# B&R Automation Studio project A2019059_Linka_Power_CP (part 13)

#### RFID.fun - Exported functions and function blocks
```iecst
FUNCTION_BLOCK TP_Init (*TODO: Add your comment here*)
	VAR_INPUT
		Enable : BOOL; (*Add your parameter comment*)
	END_VAR
	VAR_OUTPUT
		Ident : ARRAY[0..10] OF UDINT;
		Error : BOOL;
		ErrorID : UDINT;
		Busy : BOOL;
		Done : BOOL;
	END_VAR
	VAR
		StepInit : USINT;
		USBNodeListGetFuB : UsbNodeListGet;
		status : status;
		usbNodeList : ARRAY[0..31] OF UDINT;
		i : UINT;
		USBNodeGetFuB : UsbNodeGet;
		usbDevice : ARRAY[0..10] OF usbNode_typ;
		StringDevice : ARRAY[0..10] OF STRING[30];
	END_VAR
END_FUNCTION_BLOCK
(********************************************************************
 * COPYRIGHT -- Bernecker + Rainer
 ********************************************************************
 * Library: RFID
 * File: RFID.fun
 * Author: houx
 * Created: March 25, 2009
 ********************************************************************
 * Functions and function blocks of library RFID
 ********************************************************************)

FUNCTION_BLOCK TP_Info (*TODO: Add your comment here*)
	VAR_INPUT
		Enable : BOOL; (*Add your parameter comment*)
		Ident : UDINT;
	END_VAR
	VAR_OUTPUT
		Busy : BOOL;
		Done : BOOL;
		Error : BOOL;
		ErrorID : UDINT;
		Info : Info;
	END_VAR
	VAR
		Stepstatus : USINT;
		WriteData : ARRAY[0..255] OF USINT;
		FrameWriteStruct : FRM_write;
		status : status;
		FrameReadStruct : FRM_read;
		ReadBuffer : UDINT;
		ReadBufferLength : UINT;
		ReadData : ARRAY[0..255] OF USINT;
		FrameReleaseBufferStruct : FRM_rbuf;
		ID : ARRAY[0..9] OF USINT;
		StackLevel : ARRAY[0..1] OF USINT;
		KeyType : ARRAY[0..3] OF USINT;
		AN : ARRAY[0..2] OF USINT;
		sendbuffer : UDINT;
		FrameGetBufferStruct : FRM_gbuf;
		sendbufferlength : UINT;
		FrameReleaseOutputBufferStruct : FRM_robuf;
		FrameXOpenStruct : FRM_xopen;
	END_VAR
END_FUNCTION_BLOCK

FUNCTION_BLOCK TP_Unlock (*TODO: Add your comment here*)
	VAR_INPUT
		Enable : BOOL; (*Add your parameter comment*)
		Ident : UDINT;
		Data : UDINT;
	END_VAR
	VAR_OUTPUT
		Busy : BOOL;
		Error : BOOL;
		ErrorID : UDINT;
		Done : BOOL;
	END_VAR
	VAR
		StepType : USINT;
		WriteData : ARRAY[0..255] OF USINT;
		FrameWriteStruct : FRM_write;
		status : status;
		FrameReadStruct : FRM_read;
		ReadBuffer : UDINT;
		ReadBufferLength : UINT;
		ReadData : ARRAY[0..255] OF USINT;
		FrameReleaseBufferStruct : FRM_rbuf;
		string1 : STRING[20];
		string2 : STRING[10];
		CMD : UDINT;
		StepWrite : USINT;
		ERROR : ARRAY[0..2] OF USINT;
		AN : ARRAY[0..2] OF USINT;
		FrameGetBufferStruct : FRM_gbuf;
		sendbuffer : UDINT;
		sendbufferlength : UINT;
		FrameReleaseOutputBufferStruct : FRM_robuf;
		FrameXOpenStruct : FRM_xopen;
		TypeOK : BOOL;
	END_VAR
END_FUNCTION_BLOCK

FUNCTION_BLOCK TP_Lock (*TODO: Add your comment here*)
	VAR_INPUT
		Enable : BOOL; (*Add your parameter comment*)
		Ident : UDINT;
	END_VAR
	VAR_OUTPUT
		Busy : BOOL;
		ErrorID : UDINT;
		Error : BOOL;
		Done : BOOL;
	END_VAR
	VAR
		WriteData : ARRAY[0..255] OF USINT;
		FrameWriteStruct : FRM_write;
		status : status;
		FrameReadStruct : FRM_read;
		ReadBuffer : UDINT;
		ReadData : ARRAY[0..255] OF USINT;
		ReadBufferLength : UINT;
		FrameReleaseBufferStruct : FRM_rbuf;
		StepLOCK : USINT;
		AN : ARRAY[0..2] OF USINT;
		ERROR : ARRAY[0..2] OF USINT;
		TypeOK : BOOL;
		StepType : USINT;
		FrameGetBufferStruct : FRM_gbuf;
		sendbufferlength : UINT;
		sendbuffer : UDINT;
		FrameReleaseOutputBufferStruct : FRM_robuf;
		FrameXOpenStruct : FRM_xopen;
	END_VAR
END_FUNCTION_BLOCK

FUNCTION_BLOCK TP_PWProtect (*TODO: Add your comment here*)
	VAR_INPUT
		Enable : BOOL; (*Add your parameter comment*)
		Ident : UDINT;
		Data : UDINT;
	END_VAR
	VAR_OUTPUT
		Busy : BOOL;
		Error : BOOL;
		ErrorID : UDINT;
		Done : BOOL;
	END_VAR
	VAR
		TypeOK : BOOL;
		StepType : USINT;
		WriteData : ARRAY[0..255] OF USINT;
		FrameWriteStruct : FRM_write;
		status : status;
		FrameReadStruct : FRM_read;
		ReadBuffer : UDINT;
		ReadBufferLength : UINT;
		ReadData : ARRAY[0..255] OF USINT;
		FrameReleaseBufferStruct : FRM_rbuf;
		string1 : STRING[20];
		string2 : STRING[20];
		CMD : UDINT;
		StepWrite : USINT;
		AN : ARRAY[0..2] OF USINT;
		ERROR : ARRAY[0..2] OF USINT;
		FrameGetBufferStruct : FRM_gbuf;
		sendbuffer : UDINT;
		sendbufferlength : UINT;
		FrameReleaseOutputBufferStruct : FRM_robuf;
		FrameXOpenStruct : FRM_xopen;
	END_VAR
END_FUNCTION_BLOCK

FUNCTION_BLOCK TP_OnOff (*TODO: Add your comment here*)
	VAR_INPUT
		Enable : BOOL; (*Add your parameter comment*)
		Ident : UDINT;
		Mode : BOOL;
	END_VAR
	VAR_OUTPUT
		Error : BOOL;
		ErrorID : UDINT;
		Busy : BOOL;
		Done : BOOL;
	END_VAR
	VAR
		StepOnOff : USINT;
		WriteData : ARRAY[0..255] OF USINT;
		FrameWriteStruct : FRM_write;
		status : status;
		FrameReadStruct : FRM_read;
		ReadBuffer : UDINT;
		ReadBufferLength : UINT;
		ReadData : ARRAY[0..255] OF USINT;
		FrameReleaseOutputBufferStruct : FRM_robuf;
		AN : ARRAY[0..2] OF USINT;
		FrameGetBufferStruct : FRM_gbuf;
		sendbuffer : UDINT;
		sendbufferlength : UINT;
		FrameReleaseBufferStruct : FRM_rbuf;
		FrameXOpenStruct : FRM_xopen;
		FRM_close_0 : FRM_close;
	END_VAR
END_FUNCTION_BLOCK

FUNCTION_BLOCK TP_Crc (*TODO: Add your comment here*)
	VAR_INPUT
		Enable : BOOL; (*Add your parameter comment*)
		Ident : UDINT;
		Mode : BOOL;
	END_VAR
	VAR_OUTPUT
		Error : BOOL;
		ErrorID : UDINT;
		Busy : BOOL;
		Done : BOOL;
	END_VAR
	VAR
		WriteData : ARRAY[0..255] OF USINT;
		FrameWriteStruct : FRM_write;
		FrameReadStruct : FRM_read;
		ReadBuffer : UDINT;
		ReadData : ARRAY[0..255] OF USINT;
		ReadBufferLength : UINT;
		FrameReleaseBufferStruct : FRM_rbuf;
		status : status;
		StepCRC : USINT;
		AN : ARRAY[0..2] OF USINT;
		FrameGetBufferStruct : FRM_gbuf;
		sendbuffer : UDINT;
		sendbufferlength : UINT;
		FrameReleaseOutputBufferStruct : FRM_robuf;
		FrameXOpenStruct : FRM_xopen;
		FRM_close_0 : FRM_close;
	END_VAR
END_FUNCTION_BLOCK

FUNCTION_BLOCK TP_Write (*TODO: Add your comment here*)
	VAR_INPUT
		Enable : BOOL; (*Add your parameter comment*)
		RegNr : USINT;
		Data : UDINT;
		Ident : UDINT;
	END_VAR
	VAR_OUTPUT
		Busy : BOOL;
		Error : BOOL;
		ErrorID : UDINT;
		Done : BOOL;
	END_VAR
	VAR
		CMD : UDINT;
		WriteData : ARRAY[0..255] OF USINT;
		StepWrite : USINT;
		FrameWriteStruct : FRM_write;
		status : status;
		CommandReady : BOOL;
		ReadBuffer : UDINT;
		FrameReleaseBufferStruct : FRM_rbuf;
		ReadBufferLength : UINT;
		FrameReadStruct : FRM_read;
		ReadData : ARRAY[0..255] OF USINT;
		string1 : STRING[30];
		string2 : STRING[30];
		StepType : USINT;
		TypeOK : BOOL;
		string3 : STRING[10];
		AN : ARRAY[0..2] OF USINT;
		ERROR : ARRAY[0..2] OF USINT;
		KeyType : ARRAY[0..3] OF USINT;
		FrameGetBufferStruct : FRM_gbuf;
		sendbuffer : UDINT;
		sendbufferlength : UINT;
		FrameReleaseOutputBufferStruct : FRM_robuf;
		FrameXOpenStruct : FRM_xopen;
	END_VAR
END_FUNCTION_BLOCK

FUNCTION_BLOCK TP_Read (*TODO: Add your comment here*)
	VAR_INPUT
		Enable : BOOL; (*Add your parameter comment*)
		RegNr : USINT;
		Ident : UDINT;
	END_VAR
	VAR_OUTPUT
		Done : BOOL;
		Error : BOOL;
		ErrorID : UDINT;
		Busy : BOOL;
		Data : UDINT;
	END_VAR
	VAR
		CommandReady : BOOL;
		WriteData : ARRAY[0..255] OF USINT;
		status : status;
		ReadBuffer : UDINT;
		ReadBufferLength : UINT;
		ReadData : ARRAY[0..255] OF USINT;
		FrameReadStruct : FRM_read;
		data : ARRAY[0..19] OF USINT;
		FrameReleaseBufferStruct : FRM_rbuf;
		FrameWriteStruct : FRM_write;
		TypeOK : BOOL;
		StepType : USINT;
		KeyType : ARRAY[0..3] OF USINT;
		AN : ARRAY[0..2] OF USINT;
		ERROR : ARRAY[0..2] OF USINT;
		FrameGetBufferStruct : FRM_gbuf;
		sendbuffer : UDINT;
		sendbufferlength : UINT;
		FrameReleaseOutputBufferStruct : FRM_robuf;
		FrameXOpenStruct : FRM_xopen;
		StepREAD : USINT;
	END_VAR
END_FUNCTION_BLOCK
```

#### TP_Init.st
```iecst
(********************************************************************
 * COPYRIGHT -- Bernecker + Rainer
 ********************************************************************
 * Library: RFID
 * File: TP_Init.st
 * Author: houx
 * Created: March 25, 2009
 *****************************************************************
FuB: 			TP_Init
*****************************************************************
Discription:
	USB Interface:	This FuB find the Transponder Reader(USB) in the Target and read out the Interface Ident.
								Interface Ident ist required for all other FuBs in RFID Library.
								This FuB can work without any transponder in the range of Reader.
	serial Interface:	This FuB is not used to find a serial interface transponder reader
Parameter:
	Input:
		Enable(BOOL)	: The function block is only executed when enable is <> 0
	Output:
		Error(BOOL)		: Error = 0 (No Error) Error = 1(see ErrorID)
		ErrorID(UDINT)	: Number and Description in Error Table
		Busy(BOOL)		: Fub working on
		Ident(UDINT)	: Interface ID
		Done(BOOL)		: success, if TRUE
Author:	Xiaoguang Hou
		B&R Eggelsberg

History: 	V1.00.0 - 02 Sep 2008 first create
				V3.00.0 - 25 Mar 2009  update for serial interface transponder reader and created under AS3.0

*****************************************************************

 ********************************************************************
 * Implementation of library RFID
 ********************************************************************)

FUNCTION_BLOCK TP_Init

(*------------------------------------------------------	Start	---------------------------------------------------------*)
IF Enable = TRUE THEN
	IF (Done = FALSE) AND (Error = FALSE) THEN
		Busy	:=	TRUE;
		CASE StepInit OF
	(*	------------------------------------------------	search usb device	---------------------------------------------*)
			SEARCHTPLIST :
				USBNodeListGetFuB(enable := TRUE,pBuffer := ADR(usbNodeList),bufferSize := SIZEOF(usbNodeList));
				status.GetUsbList				:=USBNodeListGetFuB.status;
				IF status.GetUsbList = 0  THEN
					StepInit					:=SEARCHTP;
					USBNodeListGetFuB.enable 	:= FALSE;
				END_IF
	(*	------------------------------------------------	if Error ?show ErrorID	----------------------------------------------------*)
				IF (status.GetUsbList <> 0) AND (status.GetUsbList <> 65535) THEN
					StepInit 	:= SEARCHTPLIST;
					Error		:= TRUE;
					Busy		:= FALSE;
					ErrorID		:= status.GetUsbList;
				END_IF
	(*	----------------------------------------------- usb device identizification , a Transponder ? get the deviceID----------------------*)
			SEARCHTP:
				USBNodeGetFuB(enable := TRUE,nodeId := usbNodeList[i],pBuffer := ADR(usbDevice[i]),bufferSize :=256 (*SIZEOF(usbDevice)*));
				status.GetUsbNode := USBNodeGetFuB.status;
				IF  status.GetUsbNode = 0 THEN
					IF	(usbDevice[i].vendorId = TRANSPONDER_VENDOR_ID) AND (usbDevice[i].productId = TRANSPONDER_PRODUCT_ID) AND (usbDevice[i].bcdDevice = TRANSPONDER_BCD) THEN
						strcpy(ADR(StringDevice[i]),ADR(usbDevice[i].ifName));
						Ident[i]				:= ADR(StringDevice[i]);
						Done                    := TRUE;
						Busy                    := FALSE;
						USBNodeGetFuB.enable 	:= FALSE;
						i						:= i+1;
						IF i= USBNodeListGetFuB.listNodes THEN
							i           	        := 0;
							StepInit				:= SEARCHTPLIST;
						END_IF
					ELSE
						i						:= i+1;
					END_IF
				ELSIF status.GetUsbNode = 65535 THEN
					StepInit				:=SEARCHTP;
				ELSE
					StepInit :=  SEARCHTPLIST;
					Error 	 :=  TRUE;
					Busy     :=  FALSE;
					ErrorID  :=  status.GetUsbNode;
				END_IF
		END_CASE
	END_IF
	(*	------------------------------------------------	Not Enable, set parameters FALSE	----------------------------------------------------*)
ELSE
	Busy	:=	FALSE;
	Error	:=	FALSE;
	Done	:=	FALSE;
	ErrorID	:=	FALSE;
END_IF
(*	------------------------------------------------	end	----------------------------------------------------*)
END_FUNCTION_BLOCK
```

#### TP_Info.st
```iecst
(********************************************************************
 * COPYRIGHT -- Bernecker + Rainer
 ********************************************************************
 * Library: RFID
 * File: TP_Info.st
 * Author: houx
 * Created: March 25, 2009
*****************************************************************
FuB: 			TP_Info
;*****************************************************************
Discription:
	This FuB can be used to output the Transponder Type, the stack lever and HW/SW	versions.
	This Fub can only work, if any Transponder in the range of Reader.
	Type			: 4150 R/W or 4102 R
	Stack level		: stack level in transponder memory
	HW/SW version	:	guarantees that your application software is being operated with the correct readers.
Parameter:
			Input: 		Enable(BOOL)	:	The function block is only executed when enable is <> 0
				   			Ident(UDINT)	:	Interface Ident from TP_Init.
			Output: 	Error(BOOL)		:	Error = 0 (No Error) Error = 1(see ErrorID)
							ErrorID(UDINT)	:	Number and Description in Error Table
							Busy(BOOL)		:	if TRUE , Fub working on.
							Done(BOOL)		:	if TRUE, success
							Info(Info)		:	Structure with Type, ID and Stacklevel.
Author:				Xiaoguang Hou
							B&R Eggelsberg
;History:	V1.00.0 - 02 Sep 2008 : first create
				V3.00.0 - 25 Mar 2009 : update for serial interface transponder and created under AS3.0
 ********************************************************************
 * Implementation of library RFID
 ********************************************************************)

FUNCTION_BLOCK TP_Info
(*--------------------------------------	start	----------------------------*)
IF (Enable = 1) THEN
	IF ((Done = 0) AND (Error = 0)) THEN
		Busy	:=	TRUE;
		CASE Stepstatus OF
(*	------------------------------------------------	open the interface, get the internal Ident	----------------------------------------------------*)
			OPEN:
				FrameXOpenStruct(enable := 1,device := Ident);
				status.XOPEN 			:= FrameXOpenStruct.status;
				IF (status.XOPEN = 0) THEN
					Stepstatus          := TYPEWRITE ;
					FrameXOpenStruct.enable := FALSE;
				ELSE
					Stepstatus          := OPEN ;
					Error               := TRUE;
					ErrorID             := status.XOPEN;
					Busy                := 0;
				END_IF
			TYPEWRITE:
				memset(ADR(WriteData),0,SIZEOF(WriteData));
				strcpy(ADR(WriteData),ADR('tag,0,0,#crc$R$L'));
				FrameGetBufferStruct(enable:= 1, ident:= FrameXOpenStruct.ident);
				sendbuffer					:= FrameGetBufferStruct.buffer;
				sendbufferlength		:= FrameGetBufferStruct.buflng;
				status.GetBuffer		:= FrameGetBufferStruct.status;
				IF	(status.GetBuffer = 0)	THEN
					memcpy(sendbuffer,ADR(WriteData),sendbufferlength);
					FrameWriteStruct(enable := 1, ident := FrameXOpenStruct.ident, buffer := sendbuffer,buflng := strlen(ADR(WriteData)));
					status.WRITE 			:=	FrameWriteStruct.status;
				  	IF (status.WRITE <> 0) THEN
						FrameReleaseOutputBufferStruct(enable:=1,ident:=FrameXOpenStruct.ident,buffer:=sendbuffer,buflng:=strlen(ADR(WriteData)) );
						status.RoBuffer			:= FrameReleaseOutputBufferStruct.status;
					ELSE
				    	FrameGetBufferStruct.enable	:= 0;
						FrameWriteStruct.enable := 0;
						FrameReleaseOutputBufferStruct.enable := 0;
						Stepstatus              :=	TYPEREAD;
					END_IF
				ELSE
					ErrorID 	:= status.GetBuffer;
					Error   	:= 1;
					Busy    	:= 0;
					FrameGetBufferStruct.enable	:= 0;
					Stepstatus	:= OPEN;
				END_IF
			TYPEREAD:
				FrameReadStruct(enable:=1,ident:=FrameXOpenStruct.ident);
				ReadBuffer       	:=	FrameReadStruct.buffer;
				ReadBufferLength	:=	FrameReadStruct.buflng;
				status.READ      	:=	FrameReadStruct.status;
				IF  (status.READ = 0) THEN
					memset(ADR(ReadData),0,SIZEOF(ReadData));
					memcpy(ADR(ReadData),ReadBuffer,ReadBufferLength);                   (* copy read data into read buffer *)
					FrameReadStruct.enable	:= 0;
			        FrameReleaseBufferStruct(enable:=1, ident:=FrameXOpenStruct.ident, buffer:=ReadBuffer,buflng:=ReadBufferLength);        (* release read buffer *)
			        status.ReleaseBuffer	:=FrameReleaseBufferStruct.status;
			        IF (status.ReleaseBuffer=0) THEN
				        FrameReleaseBufferStruct.enable:=0;
						AN[0]		 :=	ReadData[0];
						AN[1]		 := ReadData[1];
						AN[2]		 := ReadData[2];
						IF	(memcmp(ADR(AN),ADR('ack'),3) = 0)	THEN
							memset(ADR(KeyType),0,SIZEOF(KeyType));
							KeyType[0]   	 := ReadData[6];
							KeyType[1] 	 := ReadData[7];
							KeyType[2] 	 := ReadData[8];
							KeyType[3] 	 := ReadData[9];
							IF (memcmp(ADR(KeyType),ADR('4150'),4) = 0) THEN
								Info.Type	:=	ADR(KeyType);
								Stepstatus	:=	IDWRITE;
							ELSIF	(memcmp(ADR(KeyType),ADR('4102'),4) = 0) THEN
								Info.Type	:=	ADR(KeyType);
								Stepstatus	:=	IDWRITE;
							ELSE
								Stepstatus	:= OPEN;
								ErrorID	:=	rfidError_tag_failed; (* unknow type of transponder *)
								Error   :=	1;
								Busy    :=	0;
							END_IF
						ELSIF	(memcmp(ADR(AN),ADR('nak'),3) = 0)	THEN
							Stepstatus	:= OPEN;
							ErrorID	:=	rfidError_tag_failed; (* negativ answer *)
							Error   :=	1;
							Busy    :=	0;
						ELSE
							Stepstatus	:= OPEN;
							ErrorID	:=	rfidError_tag_failed; (* unknow answer *)
							Error   :=	1;
							Busy    :=	0;
						END_IF
					ELSE
						Stepstatus	:=	OPEN;
						Error     	:=	1;
						ErrorID   	:=	status.ReleaseBuffer;
						Busy      	:=	0;
					END_IF
				ELSE
					memset(ADR(ReadData),0,SIZEOF(ReadData));
				END_IF
			IDWRITE:
				memset(ADR(WriteData),0,SIZEOF(WriteData));
				strcpy(ADR(WriteData),ADR('id,0,#crc$R$L'));
				FrameGetBufferStruct(enable:= 1, ident:= FrameXOpenStruct.ident);
				sendbuffer				    := FrameGetBufferStruct.buffer;
				sendbufferlength		:= FrameGetBufferStruct.buflng;
				status.GetBuffer		:= FrameGetBufferStruct.status;
				IF	(status.GetBuffer = 0)	THEN
					memcpy(sendbuffer,ADR(WriteData),sendbufferlength);
					FrameWriteStruct(enable := 1, ident := FrameXOpenStruct.ident, buffer := sendbuffer,buflng := strlen(ADR(WriteData)));
					status.WRITE 			:=	FrameWriteStruct.status;

			        IF (status.WRITE <> 0) THEN
						FrameReleaseOutputBufferStruct(enable:=1,ident:=FrameXOpenStruct.ident,buffer:=sendbuffer,buflng:= strlen(ADR(WriteData)));
						status.RoBuffer			:= FrameReleaseOutputBufferStruct.status;
						IF	(status.RoBuffer <> 0)	THEN
							ErrorID	:= status.RoBuffer;
						END_IF
					ELSE
			        	FrameWriteStruct.enable := 0;
						FrameGetBufferStruct.enable	:= 0;
						FrameReleaseOutputBufferStruct.enable := 0;
						Stepstatus              :=	IDREAD;
					END_IF
				ELSE
					ErrorID 	:= status.GetBuffer;
					Error   	:= 1;
					Busy    	:= 0;
					Stepstatus	:= OPEN;
					FrameGetBufferStruct.enable	:= 0;
				END_IF

			IDREAD:
				FrameReadStruct(enable:=1,ident:=FrameXOpenStruct.ident);
				ReadBuffer       	:=	FrameReadStruct.buffer;
				ReadBufferLength	:=	FrameReadStruct.buflng;
				status.READ      	:=	FrameReadStruct.status;
				IF  (status.READ = 0) THEN
					memset(ADR(ReadData),0,SIZEOF(ReadData));
					memcpy(ADR(ReadData),ReadBuffer,ReadBufferLength);                   (* copy read data into read buffer *)
					FrameReadStruct.enable	:=	0;
			        FrameReleaseBufferStruct(enable:=1, ident:=FrameXOpenStruct.ident, buffer:=ReadBuffer,buflng:=ReadBufferLength);        (* release read buffer *)
			        status.ReleaseBuffer	:=	FrameReleaseBufferStruct.status;
			        IF (status.ReleaseBuffer=0) THEN
				        FrameReleaseBufferStruct.enable	:=	0;
				        AN[0]	:= ReadData[0];
						AN[1]	:= ReadData[1];
						AN[2]	:= ReadData[2];
				        IF	(memcmp(ADR(AN),ADR('ack'),3) = 0) THEN
				        	memset(ADR(ID),0,SIZEOF(ID));
							ID[0] 	 	:=	ReadData[6];
							ID[1] 	 	:=	ReadData[7];
							ID[2] 	 	:=	ReadData[8];
							ID[3] 	 	:=	ReadData[9];
							ID[4] 	 	:=	ReadData[11];
							ID[5] 	 	:=	ReadData[12];
							ID[6] 	 	:=	ReadData[13];
							ID[7] 	 	:=	ReadData[14];
							Info.ID   	:=	ADR(ID);
							Stepstatus  :=	STACKWRITE;
						ELSE
							Stepstatus	:= OPEN;
							Error     	:= 1;
							ErrorID   	:= rfidError_id_failed;	(* negativ answer by ask for ID *)
							Busy      	:= 0;
						END_IF
					ELSE
						Stepstatus	:= OPEN;
						Error     	:= 1;
						ErrorID   	:= status.ReleaseBuffer;
						Busy      	:= 0;
					END_IF
				ELSE
					memset(ADR(ReadData),0,SIZEOF(ReadData));
				END_IF
			STACKWRITE:
				memset(ADR(WriteData),0,SIZEOF(WriteData));
				strcpy(ADR(WriteData),ADR('stack,0,#crc$R$L'),);
				FrameGetBufferStruct(enable:= 1, ident:= FrameXOpenStruct.ident);
				sendbuffer				:= FrameGetBufferStruct.buffer;
				sendbufferlength		:= FrameGetBufferStruct.buflng;
				status.GetBuffer		:= FrameGetBufferStruct.status;
				IF	(status.GetBuffer = 0)	THEN
					memcpy(sendbuffer,ADR(WriteData),sendbufferlength);
					FrameWriteStruct(enable := 1, ident := FrameXOpenStruct.ident, buffer := sendbuffer,buflng := strlen(ADR(WriteData)));
					status.WRITE 		:=	FrameWriteStruct.status;
			        Stepstatus          :=	STACKREAD;
			        IF (status.WRITE <> 0) THEN
						FrameReleaseOutputBufferStruct(enable:=1,ident:=FrameXOpenStruct.ident,buffer:=sendbuffer,buflng:= strlen(ADR(WriteData)));
						status.RoBuffer			:= FrameReleaseOutputBufferStruct.status;
						IF	(status.RoBuffer <> 0)	THEN
							ErrorID	:= status.RoBuffer;
						END_IF
					END_IF
					FrameWriteStruct.enable :=	0;
					FrameGetBufferStruct.enable	:= 0;
					FrameReleaseOutputBufferStruct.enable := 0;
				ELSE
					ErrorID 	:= status.GetBuffer;
					Error   	:= 1;
					Busy    	:= 0;
					Stepstatus	:= OPEN;
					FrameGetBufferStruct.enable	:= 0;
				END_IF
			STACKREAD:
				FrameReadStruct(enable:=1,ident:=FrameXOpenStruct.ident);
				ReadBuffer       	:=	FrameReadStruct.buffer;
				ReadBufferLength	:=	FrameReadStruct.buflng;
				status.READ      	:=	FrameReadStruct.status;
				IF  (status.READ = 0) THEN
					memset(ADR(ReadData),0,SIZEOF(ReadData));
					memcpy(ADR(ReadData),ReadBuffer,ReadBufferLength);                   (* copy read data into read buffer *)
					FrameReadStruct.enable	:=	0;
			        FrameReleaseBufferStruct(enable:=1, ident:=FrameXOpenStruct.ident, buffer:=ReadBuffer,buflng:=ReadBufferLength);        (* release read buffer *)
			        status.ReleaseBuffer	:=	FrameReleaseBufferStruct.status;
			        IF (status.ReleaseBuffer = 0) THEN
				        FrameReleaseBufferStruct.enable	:=	0;
				        AN[0]	:= ReadData[0];
						AN[1]	:= ReadData[1];
						AN[2]	:= ReadData[2];
				        IF	(memcmp(ADR(AN),ADR('ack'),3) = 0) THEN
							memset(ADR(StackLevel),0,SIZEOF(StackLevel));
							StackLevel[0] 	  :=	ReadData[6];
							StackLevel[1] 	  :=	ReadData[7];
							Info.StackLevel :=	ADR(StackLevel);
							Stepstatus		  :=	OPEN;
							Done			  :=	1;
							Busy			  :=	0;
						ELSE
							Stepstatus	:=	OPEN;
							Error     	:=	1;
							ErrorID   	:=	rfidError_stacklevel_failed;
							Busy      	:=	0;
						END_IF
					ELSE
						Stepstatus	:=	OPEN;
						Error     	:=	1;
						ErrorID   	:=	status.ReleaseBuffer;
						Busy      	:=	0;
					END_IF
				ELSE
					memset(ADR(ReadData),0,SIZEOF(ReadData));
				END_IF
		END_CASE
	END_IF
ELSE
	Busy    := 0;
	Error   := 0;
	ErrorID := 0;
	Done    := 0;
END_IF
END_FUNCTION_BLOCK
```

#### TP_Unlock.st
```iecst
(********************************************************************
 * COPYRIGHT -- Bernecker + Rainer
 ********************************************************************
 * Library: RFID
 * File: TP_Unlock.st
 * Author: houx
 * Created: March 25, 2009
*****************************************************************
;FuB: 			TP_Unlock
;*****************************************************************
Discription:
	This FuB is used to open a password-protected transponder so that all register can be edited.
	transponder key 4102 can not be used with this FuB.
	The password, protection word,and control word can only be modified after a valid TP_Unlock.
Parameter:
	Input:
		Enable(BOOL)	: The function block is only executed when enable is <> 0
	Output:
		Error(BOOL)		: Error = 0 (No Error) Error = 1(see ErrorID)
		ErrorID(UDINT)	: Number and Description in Error Table
		Busy(BOOL)		: Fub working on
		Ident(UDINT)	: Interface ID
		Done(BOOL)		: success, if TRUE
Author:	Xiaoguang Hou
		B&R Eggelsberg
;
;History:	V1.00.0 - 02 Sep 2008 : first create
				V3.00.0 - 25 Mar 2009 : update for serial interface transponder and created under AS3.0

 ********************************************************************
 * Implementation of library RFID
 ********************************************************************)

FUNCTION_BLOCK TP_Unlock

IF	(Enable	=	1)	THEN
	IF ((Done = 0) AND (Error = 0)) THEN
		Busy:=TRUE;
		IF TypeOK = FALSE THEN
			CASE StepType OF
(*	------------------------------------------------	open the interface, get the internal Ident	----------------------------------------------------*)
				OPEN:
					FrameXOpenStruct(enable := 1,device := Ident);
					status.XOPEN 			:= FrameXOpenStruct.status;
					IF (status.XOPEN = 0) THEN
						StepType            := WRITE ;
					ELSE
						StepType            := OPEN ;
						Error               := TRUE;
						ErrorID             := status.XOPEN;
						Busy                := 0;
					END_IF
				WRITE:
				memset(ADR(WriteData),0,SIZEOF(WriteData));
				strcpy(ADR(WriteData),ADR('tag,0,0,#crc$R$L'));
				FrameGetBufferStruct(enable:= 1, ident:= FrameXOpenStruct.ident);
				sendbuffer				:= FrameGetBufferStruct.buffer;
				sendbufferlength		:= FrameGetBufferStruct.buflng;
				status.GetBuffer		:= FrameGetBufferStruct.status;
				IF	(status.GetBuffer = 0)	THEN
					memcpy(sendbuffer,ADR(WriteData),sendbufferlength);
					FrameWriteStruct(enable := 1, ident := FrameXOpenStruct.ident, buffer := sendbuffer,buflng :=strlen(ADR(WriteData)));
					status.WRITE 				:=	FrameWriteStruct.status;
					StepType              		:=	READ;
				    IF (status.WRITE <> 0) THEN
						FrameReleaseOutputBufferStruct(enable:=1,ident:=FrameXOpenStruct.ident,buffer:=sendbuffer,buflng:=strlen(ADR(WriteData)));
						status.RoBuffer			:= FrameReleaseOutputBufferStruct.status;
						IF	(status.RoBuffer <> 0)	THEN
							ErrorID   	:= status.RoBuffer;
						END_IF
						FrameReleaseOutputBufferStruct.enable := 0;
						FrameWriteStruct.enable 	:=	0;
						FrameGetBufferStruct.enable	:=	0;
					END_IF
				ELSE
					ErrorID 	:= status.GetBuffer;
					Error   	:= 1;
					Busy    	:= 0;
					StepType	:= OPEN;
					TypeOK		:= FALSE;
					FrameGetBufferStruct.enable	:= 0;
				END_IF

				READ:
					FrameReadStruct(enable:=1,ident:=FrameXOpenStruct.ident);
					ReadBuffer       	:=	FrameReadStruct.buffer;
					ReadBufferLength	:=	FrameReadStruct.buflng;
					status.READ      	:=	FrameReadStruct.status;
					IF  (status.READ = 0) THEN
						memset(ADR(ReadData),0,SIZEOF(ReadData));
						memcpy(ADR(ReadData),ReadBuffer,ReadBufferLength);                   (* copy read data into read buffer *)
						FrameReadStruct.enable	:= 0;
				        FrameReleaseBufferStruct(enable:=1, ident:=FrameXOpenStruct.ident, buffer:=ReadBuffer,buflng:=ReadBufferLength);        (* release read buffer *)
				        status.ReleaseBuffer	:=FrameReleaseBufferStruct.status;
				        IF (status.ReleaseBuffer=0) THEN
					        FrameReleaseBufferStruct.enable:=0;
							AN[0]	:= ReadData[0];
							AN[1]	:= ReadData[1];
							AN[2]	:= ReadData[2];
							IF (memcmp(ADR(AN),ADR('ack'),3) = 0) THEN
								IF (memcmp(ADR(ReadData),ADR('ack,0,4150'),10) = 0) THEN
									StepType	:=	OPEN;
									TypeOK		:=	TRUE;
								ELSE
									StepType	:= 	OPEN;
									ErrorID		:=	rfidError_unlock_wrongType;          (*  hier ein Error difinieren soll  *)
									Error   	:=	1;
									Busy    	:=	0;
									TypeOK		:=	FALSE;
								END_IF
							ELSE
								StepType	:= 	OPEN;
								ErrorID		:=	rfidError_unlock_failed;          (*  hier ein Error difinieren soll  *)
								Error   	:=	1;
								Busy    	:=	0;
								TypeOK		:=	FALSE;
							END_IF
						ELSE
							StepType	:=	OPEN;
							Error     	:=	1;
							ErrorID   	:=	status.ReleaseBuffer;
							Busy      	:=	0;
							TypeOK		:=	FALSE;
						END_IF
					ELSE
						memset(ADR(ReadData),0,SIZEOF(ReadData));
					END_IF
			END_CASE
		END_IF
		IF	(TypeOK	= TRUE)	THEN
			string1	:=	'li,0,';
			string2	:=	',#crc$R$L';
			CMD		:=	strcat(ADR(string1),Data);
			CMD		:=	strcat(ADR(string1),ADR(string2));
			memset(ADR(WriteData),0,SIZEOF(WriteData));
			strcpy(ADR(WriteData),ADR(string1));
			CASE StepWrite OF
				OPEN:
					FrameXOpenStruct(enable := 1,device := Ident);
					status.XOPEN 			:= FrameXOpenStruct.status;
					IF (status.XOPEN = 0) THEN
						StepWrite            := WRITE ;
					ELSE
						StepWrite            := OPEN ;
						Error               := TRUE;
						ErrorID             := status.XOPEN;
						Busy                := 0;
					END_IF
				WRITE:
					FrameGetBufferStruct(enable:= 1, ident:= FrameXOpenStruct.ident);
					sendbuffer					:= FrameGetBufferStruct.buffer;
					sendbufferlength		:= FrameGetBufferStruct.buflng;
					status.GetBuffer		:= FrameGetBufferStruct.status;
					IF	(status.GetBuffer = 0)	THEN
						memcpy(sendbuffer,ADR(WriteData),sendbufferlength);
						FrameWriteStruct(enable := 1, ident := FrameXOpenStruct.ident, buffer := sendbuffer,buflng := strlen(ADR(WriteData)));
						status.WRITE 				:=	FrameWriteStruct.status;
					    IF (status.WRITE = FALSE) THEN
					    	StepWrite              		:=	READ;
							FrameWriteStruct.enable 	:=	0;
							FrameGetBufferStruct.enable	:=	0;
						ELSE
							ErrorID 				:= status.WRITE;
							Error   				:= 1;
							Busy    				:= 0;
							StepWrite				:= OPEN;
							TypeOK					:= FALSE;
							FrameWriteStruct.enable := 0;
							FrameGetBufferStruct.enable	:= 0;
							FrameReleaseOutputBufferStruct(enable:=1,ident:=FrameXOpenStruct.ident,buffer:=sendbuffer,buflng:= sendbufferlength);
							status.RoBuffer			:= FrameReleaseOutputBufferStruct.status;
							IF	(status.RoBuffer <> 0)	THEN
								StepWrite 	:= OPEN;
								Error     	:= TRUE;
								ErrorID   	:= status.RoBuffer;
								Busy      	:= 0;
								TypeOK		:= FALSE;
								FrameReleaseOutputBufferStruct.enable := 0;
							END_IF
						END_IF
					ELSE
						ErrorID 	:= status.GetBuffer;
						Error   	:= 1;
						Busy    	:= 0;
						StepWrite	:= OPEN;
						TypeOK		:= FALSE;
						FrameGetBufferStruct.enable	:= 0;
					END_IF
			    READ:
				    FrameReadStruct(enable := 1,ident:=FrameXOpenStruct.ident);
					ReadBuffer			:=	FrameReadStruct.buffer;
					ReadBufferLength	:=	FrameReadStruct.buflng;
					status.READ			:=	FrameReadStruct.status;
					IF  (status.READ = 0)  THEN
						memset(ADR(ReadData),0,SIZEOF(ReadData));
						memcpy(ADR(ReadData),ReadBuffer,ReadBufferLength);
						FrameReadStruct.enable := 0;
				        FrameReleaseBufferStruct(enable:=1, ident:=FrameXOpenStruct.ident, buffer:=ReadBuffer,buflng:=ReadBufferLength);
				        status.ReleaseBuffer	:=	FrameReleaseBufferStruct.status;
				        IF status.ReleaseBuffer=0 THEN
							FrameReleaseBufferStruct.enable:=0;
							AN[0]	:= ReadData[0];
							AN[1]	:= ReadData[1];
							AN[2]	:= ReadData[2];
							IF (memcmp(ADR(AN),ADR('ack'),3)) = 0 THEN
								StepWrite		:=	WRITE;
							 	Busy			:=	0;
							 	Done			:=	1;
								TypeOK			:=	FALSE;
							ELSIF	(memcmp(ADR(AN),ADR('nak'),3)) = 0 THEN
								ERROR[0]	:=	ReadData[6];
								ERROR[1]	:=	ReadData[7];
								ERROR[2]	:=	ReadData[8];
								Error		:=	1;
								ErrorID		:=	atoi(ADR(ERROR)) ;
								Busy		:=	0;
								TypeOK		:=	FALSE;
								StepWrite	:=	WRITE;
							ELSE
								Error			:=	1;
								ErrorID			:=	rfidError_unlock_failed ;(* unknow answer *)
								Busy			:=	0;
								TypeOK			:=	FALSE;
								StepWrite		:=	WRITE;
							END_IF
						ELSE
							Error			:=	1;
							ErrorID			:=	status.ReleaseBuffer ;
							Busy			:=	0;
							TypeOK			:=	FALSE;
							StepWrite		:=	WRITE;
					    END_IF
					ELSE
						memset(ADR(ReadData),0,SIZEOF(ReadData));
					END_IF
			END_CASE
		END_IF
	END_IF
ELSE
	Busy	:=	0;
	Error	:=	0;
	ErrorID	:=	0;
	Done	:=	0;
END_IF
END_FUNCTION_BLOCK
```

#### TP_Lock.st
```iecst
(********************************************************************
 * COPYRIGHT -- Bernecker + Rainer
 ********************************************************************
 * Library: RFID
 * File: TP_Lock.st
 * Author: houx
 * Created: March 25, 2009
 *****************************************************************
;FuB: 			TP_Lock
;*****************************************************************
Discription:
	If a password-protected transponder was opened with the TP_Unlock, it can be locked again with this FuB
	From this point on, password-protected areas can no longer be edited.
	if the transponder is removed from the reading range of the transponder reader, then it is locked automatically.
Parameter:
	Input:
		Enable(BOOL)	: The function block is only executed when enable is <> 0
	Output:
		Error(BOOL)		: Error = 0 (No Error) Error = 1(see ErrorID)
		ErrorID(UDINT)	: Number and Description in Error Table
		Busy(BOOL)		: Fub working on
		Ident(UDINT)	: Interface ID
		Done(BOOL)		: success, if TRUE
;Author:	Xiaoguang Hou
;			B&R Eggelsberg
;
;History:	V1.00.0 - 02 Sep 2008 : first create
				V3.00.0 - 25 Mar 2009 : update for serial interface transponder and created under AS3.0
;
;******************************************************************

 ********************************************************************
 * Implementation of library RFID
 ********************************************************************)
(*TODO: Add your comment here*)
FUNCTION_BLOCK TP_Lock

IF Enable = TRUE THEN
	IF ((Done = 0) AND (Error = 0)) THEN
		Busy:=TRUE;
		IF TypeOK = FALSE THEN
			CASE StepType OF
(*	------------------------------------------------	open the interface, get the internal Ident	----------------------------------------------------*)
				OPEN:
					FrameXOpenStruct(enable := 1,device := Ident);
					status.XOPEN 			:= FrameXOpenStruct.status;
					IF (status.XOPEN = 0) THEN
						StepType            := WRITE ;
					ELSE
						StepType            := OPEN ;
						Error               := TRUE;
						ErrorID             := status.XOPEN;
						Busy                := 0;
					END_IF
				WRITE:
					memset(ADR(WriteData),0,SIZEOF(WriteData));
					strcpy(ADR(WriteData),ADR('tag,0,0,#crc$R$L'));
					FrameGetBufferStruct(enable:= 1, ident:= FrameXOpenStruct.ident);
					sendbuffer				:= FrameGetBufferStruct.buffer;
					sendbufferlength		:= FrameGetBufferStruct.buflng;
					status.GetBuffer		:= FrameGetBufferStruct.status;
					IF	(status.GetBuffer = 0)	THEN
						memcpy(sendbuffer,ADR(WriteData),sendbufferlength);
						FrameWriteStruct(enable := 1, ident := FrameXOpenStruct.ident, buffer := sendbuffer,buflng := strlen(ADR(WriteData)));
						status.WRITE 				:=	FrameWriteStruct.status;
					    StepType              		:=	READ;
					    IF (status.WRITE <> 0) THEN
							FrameReleaseOutputBufferStruct(enable:=1,ident:=FrameXOpenStruct.ident,buffer:=sendbuffer,buflng:= strlen(ADR(WriteData)));
							status.RoBuffer			:= FrameReleaseOutputBufferStruct.status;
							IF	(status.RoBuffer <> 0)	THEN
								ErrorID   	:= status.RoBuffer;
							END_IF
						END_IF
						FrameWriteStruct.enable := 0;
						FrameGetBufferStruct.enable	:= 0;
						FrameReleaseOutputBufferStruct.enable := 0;
					ELSE
						ErrorID 	:= status.GetBuffer;
						Error   	:= 1;
						Busy    	:= 0;
						StepType	:= OPEN;
						TypeOK		:= FALSE;
						FrameGetBufferStruct.enable	:= 0;
					END_IF
				READ:
					FrameReadStruct(enable:=1,ident:=FrameXOpenStruct.ident);
					ReadBuffer       	:=	FrameReadStruct.buffer;
					ReadBufferLength	:=	FrameReadStruct.buflng;
					status.READ      	:=	FrameReadStruct.status;
					IF  (status.READ = 0) THEN
						memset(ADR(ReadData),0,SIZEOF(ReadData));
						memcpy(ADR(ReadData),ReadBuffer,ReadBufferLength);                   (* copy read data into read buffer *)
						FrameReadStruct.enable	:= 0;
				        FrameReleaseBufferStruct(enable:=1, ident:=FrameXOpenStruct.ident, buffer:=ReadBuffer,buflng:=ReadBufferLength);        (* release read buffer *)
				        status.ReleaseBuffer	:=FrameReleaseBufferStruct.status;
				        IF (status.ReleaseBuffer=0) THEN
					        FrameReleaseBufferStruct.enable:=0;
							AN[0]	:= ReadData[0];
							AN[1]	:= ReadData[1];
							AN[2]	:= ReadData[2];
							IF (memcmp(ADR(AN),ADR('ack'),3) = 0) THEN
								IF (memcmp(ADR(ReadData),ADR('ack,0,4150,#02d0$R$L'),SIZEOF('ack,0,4150,#02d0$R$L')) = 0) THEN
									StepType	:=	OPEN;
									TypeOK		:=	TRUE;
									StepLOCK	:=	WRITE;
								ELSE
									StepType	:= 	OPEN;
									ErrorID		:=	rfidError_lock_wrongType;          (*  hier ein Error difinieren soll  *)
									Error   	:=	1;
									Busy    	:=	0;
									TypeOK		:=	FALSE;
								END_IF
							ELSE
								StepType	:= 	OPEN;
								ErrorID		:=	rfidError_lock_failed;          (*  hier ein Error difinieren soll  *)
								Error   	:=	1;
								Busy    	:=	0;
								TypeOK		:=	FALSE;
							END_IF
						ELSE
							StepType	:=	OPEN;
							Error     	:=	1;
							ErrorID   	:=	status.ReleaseBuffer;
							Busy      	:=	0;
							TypeOK		:=	FALSE;
						END_IF
					ELSE
						memset(ADR(ReadData),0,SIZEOF(ReadData));
					END_IF
			END_CASE
		END_IF
		IF TypeOK = TRUE THEN
			CASE StepLOCK OF
				WRITE:
					memset(ADR(WriteData),0,SIZEOF(WriteData));
					strcpy(ADR(WriteData),ADR('re,0,#crc$R$L'));
					FrameGetBufferStruct(enable:= 1, ident:= FrameXOpenStruct.ident);
					sendbuffer				:= FrameGetBufferStruct.buffer;
					sendbufferlength		:= FrameGetBufferStruct.buflng;
					status.GetBuffer		:= FrameGetBufferStruct.status;
					IF	(status.GetBuffer = 0)	THEN
						memcpy(sendbuffer,ADR(WriteData),sendbufferlength);
						FrameWriteStruct(enable := 1, ident := FrameXOpenStruct.ident, buffer := sendbuffer,buflng := strlen(ADR(WriteData)));
						status.WRITE 				:=	FrameWriteStruct.status;
					   	StepLOCK              		:=	READ;
					    IF (status.WRITE <> 0) THEN
							FrameReleaseOutputBufferStruct(enable:=1,ident:=FrameXOpenStruct.ident,buffer:=sendbuffer,buflng:= sendbufferlength);
							status.RoBuffer			:= FrameReleaseOutputBufferStruct.status;
							IF	(status.RoBuffer <> 0)	THEN
								ErrorID   	:= status.RoBuffer;
							END_IF
						END_IF
						FrameWriteStruct.enable := 0;
						FrameGetBufferStruct.enable	:= 0;
						FrameReleaseOutputBufferStruct.enable := 0;
					ELSE
						ErrorID 	:= status.GetBuffer;
						Error   	:= 1;
						Busy    	:= 0;
						StepLOCK	:= WRITE;
						TypeOK		:= FALSE;
						FrameGetBufferStruct.enable	:= 0;
					END_IF
				READ:
				    FrameReadStruct(enable := 1,ident:=FrameXOpenStruct.ident);
					ReadBuffer			:= FrameReadStruct.buffer;
					ReadBufferLength	:= FrameReadStruct.buflng;
					status.READ			:= FrameReadStruct.status;
					IF  (status.READ = 0) THEN
						memset(ADR(ReadData),0,SIZEOF(ReadData));
						memcpy(ADR(ReadData),ReadBuffer,ReadBufferLength);                   (* copy read data into read buffer *)
						FrameReadStruct.enable 	:= 0;
				        FrameReleaseBufferStruct(enable:=1, ident:=FrameXOpenStruct.ident, buffer:=ReadBuffer,buflng:=ReadBufferLength);        (* release read buffer *)
				        status.ReleaseBuffer	:= FrameReleaseBufferStruct.status;
				        IF (status.ReleaseBuffer=0) THEN
						    FrameReleaseBufferStruct.enable	:= 0;
							AN[0]	:= ReadData[0];
							AN[1]	:= ReadData[1];
							AN[2]	:= ReadData[2];
							IF (memcmp(ADR(AN),ADR('ack'),3)) = 0 THEN
								StepLOCK  := WRITE;
								Done      := 1;
								Busy      := 0;
								TypeOK	  := FALSE;
							ELSIF	(memcmp(ADR(AN),ADR('nak'),3)) = 0 THEN
								ERROR[0]	:=	ReadData[6];
								ERROR[1]	:=	ReadData[7];
								ERROR[2]	:=	ReadData[8];
								Error		:=	1;
								ErrorID		:=	atoi(ADR(ERROR)) ;
								Busy		:=	0;
								TypeOK		:=	FALSE;
								StepLOCK	:=	WRITE;
							ELSE
								StepLOCK  := WRITE;
								Error     := 1;
								ErrorID   := rfidError_lock_failed; (* unknow answer *)
								Busy      := 0;
								TypeOK	  := FALSE;
							END_IF
						ELSE
							StepLOCK  := WRITE;
							Error     := 1;
							ErrorID   := status.ReleaseBuffer;
							Busy      := 0;
							TypeOK	  := FALSE;
					    END_IF
					ELSE
						memset(ADR(ReadData),0,SIZEOF(ReadData));
					END_IF
			END_CASE
		END_IF
	END_IF
ELSE
	Busy 	:= 0;
	ErrorID := 0;
	Error 	:= 0;
	Done 	:= 0;
END_IF
END_FUNCTION_BLOCK
```

#### TP_PWProtect.st
```iecst
(********************************************************************
 * COPYRIGHT -- Bernecker + Rainer
 ********************************************************************
 * Library: RFID
 * File: TP_PWProtect.st
 * Author: houx
 * Created: March 25, 2009
 *****************************************************************
;FuB: 			TP_PWProtect
;*****************************************************************
Discription:
	This FuB is used to write the password
	before a new password can be written, a valid TP_Unlock must be done.
Parameter:
	Input:
		Enable(BOOL)	:The function block is only executed when enable is <> 0
		Data(UDINT)		:Pointer to Password. whick should be write in transponder.
	Output:
		Error(BOOL)		:Error = 0 (No Error) Error = 1(see ErrorID)
		ErrorID(UDINT)	:Number and Description in Error Table
		Busy(BOOL)		:Fub working on
		Done			:success, if TRUE
;Author:	Xiaoguang Hou
;			B&R Eggelsberg
;
;History: 	V1.00.0 - 02 Sep 2008 first create
				V3.00.0 - 25 Mar 2009  update for serial interface transponder reader and created under AS3.0
;
;******************************************************************

 ********************************************************************
 * Implementation of library RFID
 ********************************************************************)

(*TODO: Add your comment here*)
FUNCTION_BLOCK TP_PWProtect

IF	(Enable	=	1)	THEN
	IF ((Done = 0) AND (Error = 0)) THEN
		Busy:=TRUE;
		IF TypeOK = FALSE THEN
			CASE StepType OF
(*	------------------------------------------------	open the interface, get the internal Ident	----------------------------------------------------*)
				OPEN:
					FrameXOpenStruct(enable := 1,device := Ident);
					status.XOPEN 			:= FrameXOpenStruct.status;
					IF (status.XOPEN = 0) THEN
						StepType            := WRITE ;
					ELSE
						StepType            := OPEN ;
						Error               := TRUE;
						ErrorID             := status.XOPEN;
						Busy                := 0;
					END_IF
				WRITE:
					memset(ADR(WriteData),0,SIZEOF(WriteData));
					strcpy(ADR(WriteData),ADR('tag,0,0,#crc$R$L'));
					FrameGetBufferStruct(enable:= 1, ident:= FrameXOpenStruct.ident);
					sendbuffer				:= FrameGetBufferStruct.buffer;
					sendbufferlength		:= FrameGetBufferStruct.buflng;
					status.GetBuffer		:= FrameGetBufferStruct.status;
					IF	(status.GetBuffer = 0)	THEN
						memcpy(sendbuffer,ADR(WriteData),sendbufferlength);
						FrameWriteStruct(enable := 1, ident := FrameXOpenStruct.ident, buffer := sendbuffer,buflng := strlen(ADR(WriteData)));
						status.WRITE 				:=	FrameWriteStruct.status;
					    StepType              		:=	READ;
					    IF (status.WRITE <> 0) THEN
							FrameReleaseOutputBufferStruct(enable:=1,ident:=FrameXOpenStruct.ident,buffer:=sendbuffer,buflng:= strlen(ADR(WriteData)));
							status.RoBuffer			:= FrameReleaseOutputBufferStruct.status;
							IF	(status.RoBuffer <> 0)	THEN
								ErrorID	:=	status.RoBuffer;
							END_IF
						END_IF
						FrameWriteStruct.enable := 0;
						FrameGetBufferStruct.enable	:= 0;
						FrameReleaseOutputBufferStruct.enable := 0;
					ELSE
						ErrorID 	:= status.GetBuffer;
						Error   	:= 1;
						Busy    	:= 0;
						StepType	:= OPEN;
						TypeOK		:= FALSE;
						FrameGetBufferStruct.enable	:= 0;
					END_IF

				READ:
					FrameReadStruct(enable:=1,ident:=FrameXOpenStruct.ident);
					ReadBuffer       	:=	FrameReadStruct.buffer;
					ReadBufferLength	:=	FrameReadStruct.buflng;
					status.READ      	:=	FrameReadStruct.status;
					IF  (status.READ = 0) THEN
						memset(ADR(ReadData),0,SIZEOF(ReadData));
						memcpy(ADR(ReadData),ReadBuffer,ReadBufferLength);                   (* copy read data into read buffer *)
						FrameReadStruct.enable	:= 0;
				        FrameReleaseBufferStruct(enable:=1, ident:=FrameXOpenStruct.ident, buffer:=ReadBuffer,buflng:=ReadBufferLength);        (* release read buffer *)
				        status.ReleaseBuffer	:=FrameReleaseBufferStruct.status;
				        IF (status.ReleaseBuffer=0) THEN
					        FrameReleaseBufferStruct.enable:=0;
							IF (memcmp(ADR(ReadData),ADR('ack,0,4150,#02d0$R$L'),SIZEOF('ack,0,4150,#02d0$R$L')) = 0) THEN
								StepType	:=	OPEN;
								TypeOK		:=	TRUE;
								StepWrite	:=	WRITE;
							ELSE
								StepType	:= 	OPEN;
								ErrorID		:=	rfidError_password_wrongType;         (*   hier ein Error difinieren soll  *)
								Error   	:=	1;
								Busy    	:=	0;
								TypeOK		:=	FALSE;
							END_IF
						ELSE
							StepType	:=	OPEN;
							Error     	:=	1;
							ErrorID   	:=	status.ReleaseBuffer;
							Busy      	:=	0;
							TypeOK		:=	FALSE;
						END_IF
					ELSE
						memset(ADR(ReadData),0,SIZEOF(ReadData));
					END_IF
			END_CASE
		END_IF
		IF	(TypeOK	= TRUE)	THEN
			string1	:=	'wp,0,';
			string2	:=	',#crc$R$L';
			CMD		:=	strcat(ADR(string1),Data);
			CMD		:=	strcat(ADR(string1),ADR(string2));
			memset(ADR(WriteData),0,SIZEOF(WriteData));
			memcpy(ADR(WriteData),ADR(string1),SIZEOF(string1));
			CASE StepWrite OF
				WRITE:
					FrameGetBufferStruct(enable:= 1, ident:= FrameXOpenStruct.ident);
					sendbuffer				:= FrameGetBufferStruct.buffer;
					sendbufferlength		:= FrameGetBufferStruct.buflng;
					status.GetBuffer		:= FrameGetBufferStruct.status;
					IF	(status.GetBuffer = 0)	THEN
						memcpy(sendbuffer,ADR(WriteData),sendbufferlength);
						FrameWriteStruct(enable := 1, ident := FrameXOpenStruct.ident, buffer := sendbuffer,buflng := strlen(ADR(WriteData)));
						status.WRITE 				:=	FrameWriteStruct.status;
					    StepWrite              		:=	READ;
					    IF (status.WRITE <> 0) THEN
							FrameReleaseOutputBufferStruct(enable:=1,ident:=FrameXOpenStruct.ident,buffer:=sendbuffer,buflng:=strlen(ADR(WriteData)) );
							status.RoBuffer			:= FrameReleaseOutputBufferStruct.status;
							IF	(status.RoBuffer <> 0)	THEN
								ErrorID	:=	status.RoBuffer;
							END_IF
						END_IF
						FrameWriteStruct.enable := 0;
						FrameGetBufferStruct.enable	:= 0;
						FrameReleaseOutputBufferStruct.enable := 0;
					ELSE
						ErrorID 	:= status.GetBuffer;
						Error   	:= 1;
						Busy    	:= 0;
						StepWrite	:= WRITE;
						TypeOK		:= FALSE;
						FrameGetBufferStruct.enable	:= 0;
					END_IF

			    READ:
				    FrameReadStruct(enable := 1,ident:=FrameXOpenStruct.ident);
					ReadBuffer			:=	FrameReadStruct.buffer;
					ReadBufferLength	:=	FrameReadStruct.buflng;
					status.READ			:=	FrameReadStruct.status;
					IF  (status.READ = 0)  THEN
						memset(ADR(ReadData),0,SIZEOF(ReadData));
						memcpy(ADR(ReadData),ReadBuffer,ReadBufferLength);
						FrameReadStruct.enable := 0;
				        FrameReleaseBufferStruct(enable:=1, ident:=FrameXOpenStruct.ident, buffer:=ReadBuffer,buflng:=ReadBufferLength);
				        status.ReleaseBuffer	:=	FrameReleaseBufferStruct.status;
				        IF status.ReleaseBuffer=0 THEN
							FrameReleaseBufferStruct.enable:=0;
							memset(ADR(AN),0,SIZEOF(AN));
							AN[0]	:= ReadData[0];
							AN[1]	:= ReadData[1];
							AN[2]	:= ReadData[2];
							IF (memcmp(ADR(AN),ADR('ack'),3)) = 0 THEN
								StepWrite		:=	WRITE;
							 	Busy			:=	0;
							 	Done			:=	1;
								TypeOK			:=	FALSE;
							ELSIF	(memcmp(ADR(AN),ADR('nak'),3)) = 0 THEN
								ERROR[0]	:=	ReadData[6];
								ERROR[1]	:=	ReadData[7];
								ERROR[2]	:=	ReadData[8];
								Error			:=	1;
								ErrorID			:=	atoi(ADR(ERROR)) ;
								Busy			:=	0;
								TypeOK			:=	FALSE;
								StepWrite		:=	WRITE;
							ELSE
								Error			:=	1;
								ErrorID			:=	rfidError_password_failed ;
								Busy			:=	0;
								TypeOK			:=	FALSE;
								StepWrite		:=	WRITE;
							END_IF
						ELSE
							Error			:=	1;
							ErrorID			:=	status.ReleaseBuffer ;
							Busy			:=	0;
							TypeOK			:=	FALSE;
							StepWrite		:=	WRITE;
					    END_IF
					ELSE
						memset(ADR(ReadData),0,SIZEOF(ReadData));
					END_IF
			END_CASE
		END_IF
	END_IF
ELSE
	Busy	:=	0;
	Error	:=	0;
	ErrorID	:=	0;
	Done	:=	0;
END_IF
END_FUNCTION_BLOCK
```

#### TP_OnOff.st
```iecst
(********************************************************************
 * COPYRIGHT -- Bernecker + Rainer
 ********************************************************************
 * Library: RFID
 * File: TP_OnOff.st
 * Author: houx
 * Created: March 25, 2009
 *****************************************************************
;FuB: 			TP_OnOff
;*****************************************************************
Discription:
	This FuB turn the 125 kHz carrier frequency of the Transponder reader/writer On/Off.
	This Fub can work without any Transponder in the range of Reader.
	Standard Configuration is frequency on.
	Be aware that no Transponder key can be read if frequency is turned off.
Parameter:
	Input:
		Enable(BOOL)	:	The function block is only executed when enable is <> 0
		Ident(UDINT)	:	Interface Ident from TP_Init.
   		Mode(BOOL)		:	frequency On:Mode=TRUE, frequency Off: Mode:=FALSE;
	Output:
		Error(BOOL)		:	Error = 0 (No Error) Error = 1(see ErrorID)
		ErrorID(UDINT)	:	Number and Description in Error Table
		Busy(BOOL)		:	if TRUE , Fub working on.
		Done(BOOL) 		:	if TRUE, success
Author:	Xiaoguang Hou
		B&R Eggelsberg

History: 	V1.00.0 - 02 Sep 2008 first create
				V3.00.0 - 25 Mar 2009  update for serial interface transponder reader and created under AS3.0

;******************************************************************

 ********************************************************************
 * Implementation of library RFID
 ********************************************************************)

(*TODO: Add your comment here*)
FUNCTION_BLOCK TP_OnOff

(*------------------------------------	Start	--------------------------------*)
IF Enable=1 THEN
	IF ((Done = 0) AND (Error = 0)) THEN
		Busy:=TRUE;
		CASE StepOnOff OF
(*	------------------------------------------------	open the interface, get the internal Ident	----------------------------------------------------*)
			OPEN:
				FrameXOpenStruct(enable := TRUE,device := Ident);
				status.XOPEN 			:= FrameXOpenStruct.status;
				IF (status.XOPEN = 0) THEN
					StepOnOff               := WRITE ;
					FrameXOpenStruct.enable:=FALSE;
				ELSE
					StepOnOff               := OPEN ;
					Error                   := TRUE;
					ErrorID                 := status.XOPEN;
					Busy                    := FALSE;
				END_IF

			WRITE:						(*------	write RF Command to	Reader	---------*)
				IF (Mode = TRUE) THEN
					memset(ADR(WriteData),0,SIZEOF(WriteData));
					strcpy(ADR(WriteData),ADR('rf,0,1,#crc$R$L'));
				ELSIF	(Mode = FALSE)	THEN
					memset(ADR(WriteData),0,SIZEOF(WriteData));
					strcpy(ADR(WriteData),ADR('rf,0,0,#crc$R$L'));
				END_IF
				(*------	get sendbuffer	---------*)
				FrameGetBufferStruct(enable:= TRUE, ident:= FrameXOpenStruct.ident);
				sendbuffer				:= FrameGetBufferStruct.buffer;
				sendbufferlength		:= FrameGetBufferStruct.buflng;
				status.GetBuffer		:= FrameGetBufferStruct.status;
				IF	(status.GetBuffer = 0)	THEN							 (*------	no error	---------*)
					memcpy(sendbuffer,ADR(WriteData),sendbufferlength);
					FrameWriteStruct(enable := TRUE, ident := FrameXOpenStruct.ident, buffer := sendbuffer,buflng :=strlen(ADR(WriteData)) );
					status.WRITE 				:=	FrameWriteStruct.status;
			        IF (status.WRITE <> 0) THEN
						FrameReleaseOutputBufferStruct(enable:=TRUE,ident:=FrameXOpenStruct.ident,buffer:=sendbuffer,buflng:= strlen(ADR(WriteData)));
						status.RoBuffer			:= FrameReleaseOutputBufferStruct.status;
						IF	(status.RoBuffer <> 0)	THEN
							ErrorID	:=	status.RoBuffer;
						END_IF
					ELSE
			        	StepOnOff              		:=	READ;
						FrameWriteStruct.enable := FALSE;
						FrameGetBufferStruct.enable	:= FALSE;
						FrameReleaseOutputBufferStruct.enable := FALSE;
					END_IF
				(*------	if get sendbuffer error	---------*)
				ELSE
					ErrorID 	:= status.GetBuffer;
					Error   	:= TRUE;
					Busy    	:= FALSE;
					StepOnOff	:= OPEN;
					FrameGetBufferStruct.enable	:= FALSE;
				END_IF

	    	READ:						(*	read out the feedback	*)
			    FrameReadStruct(enable := 1,ident:=FrameXOpenStruct.ident);
				ReadBuffer				:=FrameReadStruct.buffer;
				ReadBufferLength		:=FrameReadStruct.buflng;
				status.READ				:=FrameReadStruct.status;
				IF  (status.READ = 0) THEN
					memset(ADR(ReadData),0,SIZEOF(ReadData));
					memcpy(ADR(ReadData),ReadBuffer,ReadBufferLength);	(*	copy the answer	out in ReadData	*)
					FrameReadStruct.enable := 0;
			        FrameReleaseBufferStruct(enable:=1, ident:=FrameXOpenStruct.ident, buffer:=ReadBuffer,buflng:=ReadBufferLength);	(*	release the buffer	*)
			        status.ReleaseBuffer   := FrameReleaseBufferStruct.status;
			        IF (status.ReleaseBuffer=0) THEN
			        	FrameReleaseBufferStruct.enable	:= 0;
			        	AN[0]	:= ReadData[0];
						AN[1]	:= ReadData[1];
						AN[2]	:= ReadData[2];
						IF (memcmp(ADR(AN),ADR('ack'),3) = 0) THEN				(*--- positiv answer ----*)
							StepOnOff   := CLOSE;
						ELSE
							StepOnOff   := OPEN;								(*	negativ answer or unknow answer	*)
							Error     	:= 1;
							ErrorID   	:= rfidError_rf_failed;
							Busy      	:= 0;
						END_IF
					ELSE														(*	if buffer release error	*)
							StepOnOff   := OPEN;
							Error     	:= 1;
							ErrorID   	:= status.ReleaseBuffer;
							Busy     	:= 0;
			        END_IF
				ELSE
					memset(ADR(ReadData),0,SIZEOF(ReadData));
				END_IF
			CLOSE:
				FRM_close_0(enable :=1 , ident :=FrameXOpenStruct.ident);
				IF FRM_close_0.status=FALSE THEN
					Done      	:= 1;
					Busy      	:= 0;
					StepOnOff:=OPEN;
				END_IF
		END_CASE
	END_IF
ELSE                                          (*------- if enable = False ,then all output variable back to zero -------*)
	Error:=0;
	ErrorID:=0;
	Busy:=0;
	Done:=0;
END_IF
END_FUNCTION_BLOCK
```

#### TP_Crc.st
```iecst
(********************************************************************
 * COPYRIGHT -- Bernecker + Rainer
 ********************************************************************
 * Library: RFID
 * File: TP_Crc.st
 * Author: houx
 * Created: March 25, 2009
*****************************************************************
;FuB: 			TP_CRC
;*****************************************************************
Discription:
	This FuB can specify whether the transponder reader should check the checksum wenn a command string is received.
	This Fub can work without any Transponder in the range of Reader.
Parameter:
	Input: 	Enable(BOOL)	: The function block is only executed when enable is <> 0.
			Ident(UDINT)	: Interface Ident.
			Mode(BOOL)		: checksum On:Mode=TRUE, checksum Off: Mode:=FALSE;
	Output: Error(BOOL)		: Error = 0 (No Error) Error = 1(see ErrorID).
			ErrorID(UDINT)	: Number and description in error table.
			Busy(BOOL)		: FuB is working on.
			Done(BOOL)		: if TRUE, success.
Author:	Xiaoguang Hou
		B&R Eggelsberg

History: 	V1.00.0 - 02 Sep 2008 first create
				V3.00.0 - 25 Mar 2009  update for serial interface transponder readerand created under AS3.0
;
;******************************************************************

 ********************************************************************
 * Implementation of library RFID
 ********************************************************************)

(*TODO: Add your comment here*)
FUNCTION_BLOCK TP_Crc

IF Enable=1 THEN
	IF ((Done = 0) AND (Error = 0)) THEN
		Busy:=TRUE;
		CASE StepCRC OF
(*	------------------------------------------------	open the interface, get the internal Ident	----------------------------------------------------*)
			OPEN:
				FrameXOpenStruct(enable := 1,device := Ident);
				status.XOPEN 			:= FrameXOpenStruct.status;
				IF (status.XOPEN = 0) THEN
					StepCRC             := WRITE ;
					FrameXOpenStruct.enable:=FALSE;
				ELSE
					StepCRC             := OPEN ;
					Error               := TRUE;
					ErrorID             := status.XOPEN;
					Busy                := 0;
				END_IF
			WRITE:
				IF 	(Mode = TRUE) THEN
					memset(ADR(WriteData),0,SIZEOF(WriteData));
					strcpy(ADR(WriteData),ADR('cc,0,1,#01ce$R$L'));
				ELSIF (Mode = FALSE) THEN
					memset(ADR(WriteData),0,SIZEOF(WriteData));
					strcpy(ADR(WriteData),ADR('cc,0,0,#01cd$R$L'));
				END_IF
				FrameGetBufferStruct(enable:= 1, ident:= FrameXOpenStruct.ident);
				sendbuffer				:= FrameGetBufferStruct.buffer;
				sendbufferlength		:= FrameGetBufferStruct.buflng;
				status.GetBuffer		:= FrameGetBufferStruct.status;
				IF	(status.GetBuffer = 0)	THEN
					memcpy(sendbuffer,ADR(WriteData),sendbufferlength);
					FrameWriteStruct(enable := 1, ident := FrameXOpenStruct.ident, buffer := sendbuffer, buflng := strlen(ADR(WriteData)));
					status.WRITE 				:=	FrameWriteStruct.status;

			    	IF (status.WRITE <> 0) THEN
						FrameReleaseOutputBufferStruct(enable:=1,ident:=FrameXOpenStruct.ident,buffer:=sendbuffer,buflng:= strlen(ADR(WriteData)));
						status.RoBuffer			:= FrameReleaseOutputBufferStruct.status;
						IF	(status.RoBuffer <> 0)	THEN
							ErrorID:=status.RoBuffer;
						END_IF
					ELSE
			   			FrameWriteStruct.enable := 0;
						FrameGetBufferStruct.enable	:= 0;
						FrameReleaseOutputBufferStruct.enable := 0;
						StepCRC					:= READ;
					END_IF
				ELSE
					ErrorID 	:= status.GetBuffer;
					Error   	:= 1;
					Busy    	:= 0;
					StepCRC		:= OPEN;
					FrameGetBufferStruct.enable	:= 0;
				END_IF

		    READ:
			    FrameReadStruct(enable := 1,ident:=FrameXOpenStruct.ident);
				ReadBuffer			:= FrameReadStruct.buffer;
				ReadBufferLength	:= FrameReadStruct.buflng;
				status.READ			:= FrameReadStruct.status;
				IF  (status.READ = 0) THEN
					memset(ADR(ReadData),0,SIZEOF(ReadData));
					memcpy(ADR(ReadData),ReadBuffer,ReadBufferLength);                   (* copy read data into read buffer *)
					FrameReadStruct.enable 	:= 0;
			        FrameReleaseBufferStruct(enable:=1, ident:=FrameXOpenStruct.ident, buffer:=ReadBuffer,buflng:=ReadBufferLength);        (* release read buffer *)
			        status.ReleaseBuffer	:= FrameReleaseBufferStruct.status;
			        IF (status.ReleaseBuffer=0) THEN
				        FrameReleaseBufferStruct.enable	:=0;
		        		AN[0]	:= ReadData[0];
						AN[1]	:= ReadData[1];
						AN[2]	:= ReadData[2];
						IF (memcmp(ADR(AN),ADR('ack'),3) = 0) THEN
							StepCRC   := CLOSE;
						ELSE
							StepCRC   := OPEN;
							Error     := 1;
							ErrorID   := rfidError_crc_failed; (*	negativ answer *)
							Busy      := 0;
						END_IF
					ELSE
							StepCRC   := OPEN;
							Error     := 1;
							ErrorID   := status.ReleaseBuffer;
							Busy      := 0;
			        END_IF
				ELSE
					memset(ADR(ReadData),0,SIZEOF(ReadData));
				END_IF
			CLOSE:
				FRM_close_0(enable :=1 , ident :=FrameXOpenStruct.ident);
				IF FRM_close_0.status=FALSE  THEN
					Done      := 1;
					Busy      := 0;
					StepCRC   := OPEN;
				END_IF
		END_CASE
	END_IF
ELSE
	Error   := 0;
	ErrorID := 0;
	Busy    := 0;
	Done    := 0;
END_IF

END_FUNCTION_BLOCK
```

#### TP_Write.st
```iecst
(********************************************************************
 * COPYRIGHT -- Bernecker + Rainer
 ********************************************************************
 * Library: RFID
 * File: TP_Write.st
 * Author: houx
 * Created: March 25, 2009
 ****************************************************************
;FuB: 			TP_Write
;*****************************************************************
Discription:
	This FuB is used to write the registers of the transponder.
	for this to work, the transponder must not be password-protected or a valid TP_unlock must be carried out beforehand.
	Be aware that Register 1 and 2 of TP 4150 are used for the control and protectionwords.
	Only modify these registers,if you are familiar with their Function. In addition, avalid login is needed.
Parameter:
	Input:
		Enable(BOOL)	: The function block is only executed when enable is <> 0
		RegNr(USINT)	: Number of the register, which should be write in
		Data(UDINT)		: pointer to input Data
	Output:
		Error(BOOL)		: Error = 0 (No Error) Error = 1(see ErrorID)
		ErrorID(UDINT)	: Number and Description in Error Table
		Busy(BOOL)		: Fub working on
		Ident(UDINT)	: Interface ID
		Done(BOOL)		:success, if TRUE
Author:	Xiaoguang Hou
		B&R Eggelsberg
;
History: 	V1.00.0 - 02 Sep 2008 first create
				V3.00.0 - 25 Mar 2009  update for serial interface transponder reader and created under AS3.0
;
 ********************************************************************
 * Implementation of library RFID
 ********************************************************************)

(*TODO: Add your comment here*)
FUNCTION_BLOCK TP_Write

IF (Enable = 1) THEN
	IF ((Done = 0) AND (Error = 0)) THEN
		Busy:=TRUE;
		IF TypeOK = FALSE THEN
			CASE StepType OF
(*	------------------------------------------------	open the interface, get the internal Ident	----------------------------------------------------*)
				OPEN:
					FrameXOpenStruct(enable := 1,device := Ident);
					status.XOPEN 			:= FrameXOpenStruct.status;
					IF (status.XOPEN = 0) THEN
						StepType            := WRITE ;
					ELSE
						StepType            := OPEN ;
						Error               := TRUE;
						ErrorID             := status.XOPEN;
						Busy                := 0;
					END_IF
				WRITE:
					memset(ADR(WriteData),0,SIZEOF(WriteData));
					strcpy(ADR(WriteData),ADR('tag,0,0,#crc$R$L'));
					FrameGetBufferStruct(enable:= 1, ident:= FrameXOpenStruct.ident);
					sendbuffer				:= FrameGetBufferStruct.buffer;
					sendbufferlength		:= FrameGetBufferStruct.buflng;
					status.GetBuffer		:= FrameGetBufferStruct.status;
					IF	(status.GetBuffer = 0)	THEN
						memcpy(sendbuffer,ADR(WriteData),sendbufferlength);
						FrameWriteStruct(enable := 1, ident := FrameXOpenStruct.ident, buffer := sendbuffer,buflng := strlen(ADR(WriteData)));
						status.WRITE 				:=	FrameWriteStruct.status;
						StepType				:= READ;
					    IF (status.WRITE <> 0) THEN
							FrameReleaseOutputBufferStruct(enable:=1,ident:=FrameXOpenStruct.ident,buffer:=sendbuffer,buflng:= strlen(ADR(WriteData)));
							status.RoBuffer			:= FrameReleaseOutputBufferStruct.status;
							IF	(status.RoBuffer <> 0)	THEN
								ErrorID	:=	status.RoBuffer;
							END_IF
						END_IF
						FrameWriteStruct.enable := 0;
						FrameGetBufferStruct.enable	:= 0;
						FrameReleaseOutputBufferStruct.enable := 0;
					ELSE
						ErrorID 	:= status.GetBuffer;
						Error   	:= 1;
						Busy    	:= 0;
						StepType	:= OPEN;
						TypeOK		:= FALSE;
						FrameGetBufferStruct.enable	:= 0;
					END_IF

				READ:
					FrameReadStruct(enable:=1,ident:=FrameXOpenStruct.ident);
					ReadBuffer       	:=	FrameReadStruct.buffer;
					ReadBufferLength	:=	FrameReadStruct.buflng;
					status.READ      	:=	FrameReadStruct.status;
					IF  (status.READ = 0) THEN
						memset(ADR(ReadData),0,SIZEOF(ReadData));
						memcpy(ADR(ReadData),ReadBuffer,ReadBufferLength);                   (* copy read data into read buffer *)
						FrameReadStruct.enable	:= 0;
				        FrameReleaseBufferStruct(enable:=1, ident:=FrameXOpenStruct.ident, buffer:=ReadBuffer,buflng:=ReadBufferLength);        (* release read buffer *)
				        status.ReleaseBuffer	:=FrameReleaseBufferStruct.status;
				        IF (status.ReleaseBuffer=0) THEN
					        FrameReleaseBufferStruct.enable:=0;
							AN[0]		 :=	ReadData[0];
							AN[1]		 := ReadData[1];
							AN[2]		 := ReadData[2];
							IF	(memcmp(ADR(AN),ADR('ack'),3) = 0)	THEN
								memset(ADR(KeyType),0,SIZEOF(KeyType));
								KeyType[0] 	 :=	ReadData[6];
								KeyType[1] 	 := ReadData[7];
								KeyType[2] 	 := ReadData[8];
								KeyType[3] 	 := ReadData[9];
								IF (memcmp(ADR(KeyType),ADR('4150'),4) = 0) THEN
									StepType	:=	OPEN;
									TypeOK		:=	TRUE;
								ELSIF	(memcmp(ADR(KeyType),ADR('4102'),4) = 0) THEN
									StepType	:= 	OPEN;
									ErrorID		:=	rfidError_write_wrongType;         (*   wrong Type *)
									Error   	:=	1;
									Busy    	:=	0;
									TypeOK		:=	FALSE;
								ELSE
									StepType		:= 	OPEN;
									ErrorID			:=	rfidError_write_wrongType;            (* unknow type to write  *)
									Error   		:=	1;
									Busy    		:=	0;
									TypeOK			:=	FALSE;
								END_IF
							ELSIF	(memcmp(ADR(AN),ADR('nak'),3) = 0)	THEN
								StepType		:=	OPEN;
								ErrorID			:=	rfidError_write_failed; (* negativ answer *)
								Error   		:=	1;
								Busy    		:=	0;
								TypeOK			:=	FALSE;
							ELSE
								StepType	:= 	OPEN;
								ErrorID		:=	rfidError_write_failed; (* unknow answer *)
								Error   	:=	1;
								Busy    	:=	0;
								TypeOK			:=	FALSE;
							END_IF
						ELSE
							StepType	:=	OPEN;
							Error     	:=	1;
							ErrorID   	:=	status.ReleaseBuffer;
							Busy      	:=	0;
							TypeOK		:=	FALSE;
						END_IF
					ELSE
						memset(ADR(ReadData),0,SIZEOF(ReadData));
					END_IF
			END_CASE
		END_IF
		IF	(TypeOK	= TRUE)	THEN
			IF	(CommandReady = 0) THEN
				IF	(RegNr > 31) THEN
					Error	:=	1;
					ErrorID	:=	rfidError_write_wrongRegNr; (* hier soll ein Fehler Meldung difiniert werden: password Register, please use TP_Password Fub*)
					Busy	:=	0;
					TypeOK	:=	FALSE;
				ELSE
					itoa(RegNr,ADR(string1));
					string2:='wr,0,';
					string3:=',#crc$R$L';
					CMD	:=	strcat(ADR(string2),ADR(string1));
					CMD	:=	strcat(ADR(string2),ADR(','));
					CMD	:=	strcat(ADR(string2),Data);
					CMD	:=	strcat(ADR(string2),ADR(string3));
					memset(ADR(WriteData),0,SIZEOF(WriteData));
					strcpy(ADR(WriteData),ADR(string2));
					CommandReady:=	1;
					StepWrite	:=	WRITE;
				END_IF
			ELSE
				CASE StepWrite OF
					WRITE:
						FrameGetBufferStruct(enable:= 1, ident:= FrameXOpenStruct.ident);
						sendbuffer				:= FrameGetBufferStruct.buffer;
						sendbufferlength		:= FrameGetBufferStruct.buflng;
						status.GetBuffer		:= FrameGetBufferStruct.status;
						IF	(status.GetBuffer = 0)	THEN
							memcpy(sendbuffer,ADR(WriteData),sendbufferlength);
							FrameWriteStruct(enable := 1, ident := FrameXOpenStruct.ident, buffer := sendbuffer,buflng := strlen(ADR(WriteData)));
							status.WRITE 				:=	FrameWriteStruct.status;
						    StepWrite              		:=	READ;
						    IF (status.WRITE <> 0) THEN
								FrameReleaseOutputBufferStruct(enable:=1,ident:=FrameXOpenStruct.ident,buffer:=sendbuffer,buflng:= strlen(ADR(WriteData)));
								status.RoBuffer			:= FrameReleaseOutputBufferStruct.status;
								IF	(status.RoBuffer <> 0)	THEN
									ErrorID	:=	status.RoBuffer;
								END_IF
							END_IF
							FrameWriteStruct.enable := 0;
							FrameGetBufferStruct.enable	:= 0;
							FrameReleaseOutputBufferStruct.enable := 0;
						ELSE
							ErrorID 		:= status.GetBuffer;
							Error   		:= 1;
							Busy    		:= 0;
							StepWrite		:= WRITE;
							TypeOK			:= FALSE;
							CommandReady	:=	0;
							FrameGetBufferStruct.enable	:= 0;
						END_IF

			    	READ:
				    	FrameReadStruct(enable := 1,ident:=FrameXOpenStruct.ident);
						ReadBuffer			:=	FrameReadStruct.buffer;
						ReadBufferLength	:=	FrameReadStruct.buflng;
						status.READ			:=	FrameReadStruct.status;
						IF  (status.READ = 0)  THEN
							memset(ADR(ReadData),0,SIZEOF(ReadData));
							memcpy(ADR(ReadData),ReadBuffer,ReadBufferLength);
							FrameReadStruct.enable := 0;
					        FrameReleaseBufferStruct(enable:=1, ident:=FrameXOpenStruct.ident, buffer:=ReadBuffer,buflng:=ReadBufferLength);
					        status.ReleaseBuffer	:=	FrameReleaseBufferStruct.status;
					        IF status.ReleaseBuffer=0 THEN
								FrameReleaseBufferStruct.enable:=0;
					        	AN[0]	:= ReadData[0];
								AN[1]	:= ReadData[1];
								AN[2]	:= ReadData[2];
								IF (memcmp(ADR(AN),ADR('ack'),3) = 0) THEN
									StepWrite		:=	WRITE;
								 	Busy			:=	0;
								 	Done			:=	1;
									CommandReady	:=	0;
									TypeOK			:=	FALSE;
								ELSIF	(memcmp(ADR(AN),ADR('nak'),3) = 0)	THEN
									ERROR[0]	:=	ReadData[6];
									ERROR[1]	:=	ReadData[7];
									ERROR[2]	:=	ReadData[8];
									Error			:=	1;
									ErrorID			:=	rfidError_write_failed ;
									Busy			:=	0;
									CommandReady	:=	0;
									TypeOK			:=	FALSE;
									StepWrite		:=	WRITE;
								ELSE
									Error			:=	1;
									ErrorID			:=	rfidError_write_failed;
									Busy			:=	0;
									CommandReady	:=	0;
									TypeOK			:=	FALSE;
									StepWrite		:=	WRITE;
								END_IF
							ELSE
								Error			:=	1;
								ErrorID			:=	status.ReleaseBuffer ;
								Busy			:=	0;
								CommandReady	:=	0;
								TypeOK			:=	FALSE;
								StepWrite		:=	WRITE;
					       	END_IF
						ELSE
							memset(ADR(ReadData),0,SIZEOF(ReadData));
						END_IF
				END_CASE
			END_IF
		END_IF
	END_IF
ELSE
	Busy	:= 0;
	Error   := 0;
	ErrorID := 0;
	Done	:= 0;
END_IF
END_FUNCTION_BLOCK
```

#### TP_Read.st
```iecst
(********************************************************************
 * COPYRIGHT -- Bernecker + Rainer
 ********************************************************************
 * Library: RFID
 * File: TP_Read.st
 * Author: houx
 * Created: March 25, 2009
 *****************************************************************
;FuB: 			TP_Read
;*****************************************************************
Discription:
	This FuB is used to read the registers of the transponder.
	for this to work, the transponder must not be password-protected or a valid TP_unlock needs to be performed beforehand.
Parameter:
	Input:
		Enable(BOOL)	: The function block is only executed when enable is <> 0
		RegNr(USINT)	: Number of the register, which should be read out
	Output:
		Error(BOOL)		: Error = 0 (No Error) Error = 1(see ErrorID)
		ErrorID(BOOL)	: Number and Description in Error Table
		Busy(BOOL)		: Fub working on
		Data(BOOL)		: pointer to output Data.
		Done(BOOL)		: success, if TRUE
Author:	Xiaoguang Hou
		B&R Eggelsberg

History: 	V1.00.0 - 02 Sep 2008 first create
				V3.00.0 - 25 Mar 2009  update for serial interface transponder reader and created under AS3.0

 ********************************************************************
 * Implementation of library RFID
 ********************************************************************)

(*TODO: Add your comment here*)
FUNCTION_BLOCK TP_Read

    IF Enable = TRUE THEN
        IF ((Done = 0) AND (Error = 0)) THEN
            Busy:=TRUE;
            IF (TypeOK = FALSE) THEN
                CASE StepType OF
                    (*	------------------------------------------------	open the interface, get the internal Ident	----------------------------------------------------*)
                    OPEN:
                        FrameXOpenStruct.mode:=ADR(' /RIT=200 ');			(* long receive idle time for receive the data*)
                        FrameXOpenStruct(enable := 1,device := Ident);
                        status.XOPEN 			:= FrameXOpenStruct.status;
                        IF (status.XOPEN = 0) THEN
                            StepType            := WRITE ;
                            FrameXOpenStruct.enable := 0;
                        ELSE
                            StepType            := OPEN ;
                            Error               := TRUE;
                            ErrorID             := status.XOPEN;
                            Busy                := 0;
                            FrameXOpenStruct.enable := 0;
                        END_IF
                    WRITE:
                        memset(ADR(WriteData),0,SIZEOF(WriteData));
                        strcpy(ADR(WriteData),ADR('tag,0,#crc$R$L'));
                        FrameGetBufferStruct(enable:= 1, ident:= FrameXOpenStruct.ident);
                        sendbuffer					:= FrameGetBufferStruct.buffer;
                        sendbufferlength		:= FrameGetBufferStruct.buflng;
                        status.GetBuffer		:= FrameGetBufferStruct.status;
                        IF	(status.GetBuffer = 0)	THEN
                            memcpy(sendbuffer,ADR(WriteData),sendbufferlength);
                            FrameWriteStruct(enable := 1, ident := FrameXOpenStruct.ident, buffer := sendbuffer,buflng := strlen(ADR(WriteData)) );
                            status.WRITE 				:=	FrameWriteStruct.status;
                            IF (status.WRITE <> 0) THEN
                                FrameReleaseOutputBufferStruct(enable:=1,ident:=FrameXOpenStruct.ident,buffer:=sendbuffer,buflng:= strlen(ADR(WriteData)));
                                status.RoBuffer				:= FrameReleaseOutputBufferStruct.status;
                                IF (status.RoBuffer <> 0) THEN
                                    ErrorID:=status.RoBuffer;
                                END_IF
                            ELSE
                                StepType	:=	READ;
                                FrameWriteStruct.enable 	:= 0;
                                FrameGetBufferStruct.enable	:= 0;
                                FrameReleaseOutputBufferStruct.enable := 0;
                            END_IF
                        ELSE
                            ErrorID 	:= status.GetBuffer;
                            Error   	:= 1;
                            Busy    	:= 0;
                            StepType	:= OPEN;
                            TypeOK		:= FALSE;
                            FrameGetBufferStruct.enable	:= 0;
                        END_IF
                    READ:
                        FrameReadStruct(enable:=1,ident:=FrameXOpenStruct.ident);
                        ReadBuffer       	:=	FrameReadStruct.buffer;
                        ReadBufferLength	:=	FrameReadStruct.buflng;
                        status.READ      	:=	FrameReadStruct.status;
                        IF  (status.READ = 0) THEN
                            memset(ADR(ReadData),0,SIZEOF(ReadData));
                            memcpy(ADR(ReadData),ReadBuffer,ReadBufferLength);                   (* copy read data into read buffer *)
                            FrameReadStruct.enable	:= 0;
                            FrameReleaseBufferStruct(enable:=1, ident:=FrameXOpenStruct.ident, buffer:=ReadBuffer,buflng:=ReadBufferLength);        (* release read buffer *)
                            status.ReleaseBuffer	:=FrameReleaseBufferStruct.status;
                            IF (status.ReleaseBuffer=0) THEN
                                FrameReleaseBufferStruct.enable:=0;
                                AN[0]		 := ReadData[0];
                                AN[1]		 := ReadData[1];
                                AN[2]		 := ReadData[2];
                                IF	(memcmp(ADR(AN),ADR('ack'),3) = 0)	THEN
                                    memset(ADR(KeyType),0,SIZEOF(KeyType));
                                    KeyType[0] 	 := ReadData[6];
                                    KeyType[1] 	 := ReadData[7];
                                    KeyType[2] 	 := ReadData[8];
                                    KeyType[3] 	 := ReadData[9];
                                    IF (memcmp(ADR(KeyType),ADR('4150'),4) = 0) THEN
                                        StepType		:=	OPEN;
                                        Done         	:=	FALSE;
                                        Busy         	:=	0;
                                        CommandReady	:=	0;
                                        TypeOK			:=	TRUE;
                                    ELSIF	(memcmp(ADR(KeyType),ADR('4102'),4) = 0) THEN
                                        memset(ADR(data),0,SIZEOF(data));
                                        data[0] 	 	:=	ReadData[11];
                                        data[1] 	 	:=	ReadData[12];
                                        data[2] 	 	:=	ReadData[13];
                                        data[3] 	 	:=	ReadData[14];
                                        data[4] 	 	:=	ReadData[15];
                                        data[5] 	 	:=	ReadData[16];
                                        data[6] 	 	:=	ReadData[17];
                                        data[7] 	 	:=	ReadData[18];
                                        data[8] 	 	:=	ReadData[19];
                                        data[9] 	 	:=	ReadData[20];
                                        Data			:=	ADR(data);
                                        StepType		:=	OPEN;
                                        Done         	:=	1;
                                        Busy         	:=	0;
                                        CommandReady	:=	0;
                                        TypeOK			:=	FALSE;
                                    ELSE
                                        StepType		:= 	OPEN;
                                        ErrorID			:=	rfidError_read_wrongType;            (* wrong type to read  *)
                                        Error   		:=	1;
                                        Busy    		:=	0;
                                        CommandReady	:=	0;
                                        TypeOK			:=	FALSE;
                                    END_IF
                                ELSIF	(memcmp(ADR(AN),ADR('nak'),3) = 0)	THEN
                                    StepType		:= 	OPEN;
                                    ErrorID			:=	rfidError_read_failed; (* negativ answer *)
                                    Error   		:=	1;
                                    Busy    		:=	0;
                                    CommandReady	:=	0;
                                    TypeOK			:=	FALSE;
                                ELSE
                                    StepType		:=	OPEN;
                                    ErrorID			:=	rfidError_read_failed; (* unknow answer *)
                                    Error   		:=	1;
                                    Busy    		:=	0;
                                    CommandReady	:=	0;
                                    TypeOK			:=	FALSE;
                                END_IF
                            ELSE
                                StepType		:=	OPEN;
                                Error     		:=	1;
                                ErrorID   		:=	status.ReleaseBuffer;
                                Busy      		:=	0;
                                CommandReady	:=	0;
                                TypeOK			:=	FALSE;
                            END_IF
                        ELSE
                            memset(ADR(ReadData),0,SIZEOF(ReadData));
                        END_IF
                END_CASE
            END_IF
            IF	(TypeOK = TRUE) THEN
                IF CommandReady = 0 THEN
                    IF  ((0 < RegNr) AND (RegNr <34)) THEN
                        memset(ADR(WriteData),0,SIZEOF(WriteData));
                        CASE RegNr OF
                            REG1:
                                strcpy(ADR(WriteData),ADR('rdm,0,1,1,#crc$R$L'));
                            REG2:
                                strcpy(ADR(WriteData),ADR('rdm,0,2,1,#crc$R$L'));
                            REG3:
                                strcpy(ADR(WriteData),ADR('rdm,0,3,1,#crc$R$L'));
                            REG4:
                                strcpy(ADR(WriteData),ADR('rdm,0,4,1,#crc$R$L'));
                            REG5:
                                strcpy(ADR(WriteData),ADR('rdm,0,5,1,#crc$R$L'));
                            REG6:
                                strcpy(ADR(WriteData),ADR('rdm,0,6,1,#crc$R$L'));
                            REG7:
                                strcpy(ADR(WriteData),ADR('rdm,0,7,1,#crc$R$L'));
                            REG8:
                                strcpy(ADR(WriteData),ADR('rdm,0,8,1,#crc$R$L'));
                            REG9:
                                strcpy(ADR(WriteData),ADR('rdm,0,9,1,#crc$R$L'));
                            REG10:
                                strcpy(ADR(WriteData),ADR('rdm,0,10,1,#crc$R$L'));
                            REG11:
                                strcpy(ADR(WriteData),ADR('rdm,0,11,1,#crc$R$L'));
                            REG12:
                                strcpy(ADR(WriteData),ADR('rdm,0,12,1,#crc$R$L'));
                            REG13:
                                strcpy(ADR(WriteData),ADR('rdm,0,13,1,#crc$R$L'));
                            REG14:
                                strcpy(ADR(WriteData),ADR('rdm,0,14,1,#crc$R$L'));
                            REG15:
                                strcpy(ADR(WriteData),ADR('rdm,0,15,1,#crc$R$L'));
                            REG16:
                                strcpy(ADR(WriteData),ADR('rdm,0,16,1,#crc$R$L'));
                            REG17:
                                strcpy(ADR(WriteData),ADR('rdm,0,17,1,#crc$R$L'));
                            REG18:
                                strcpy(ADR(WriteData),ADR('rdm,0,18,1,#crc$R$L'));
                            REG19:
                                strcpy(ADR(WriteData),ADR('rdm,0,19,1,#crc$R$L'));
                            REG20:
                                strcpy(ADR(WriteData),ADR('rdm,0,20,1.#crc$R$L'));
                            REG21:
                                strcpy(ADR(WriteData),ADR('rdm,0,21,1,#crc$R$L'));
                            REG22:
                                strcpy(ADR(WriteData),ADR('rdm,0,22,1,#crc$R$L'));
                            REG23:
                                strcpy(ADR(WriteData),ADR('rdm,0,23,1,#crc$R$L'));
                            REG24:
                                strcpy(ADR(WriteData),ADR('rdm,0,24,1,#crc$R$L'));
                            REG25:
                                strcpy(ADR(WriteData),ADR('rdm,0,25,1,#crc$R$L'));
                            REG26:
                                strcpy(ADR(WriteData),ADR('rdm,0,26,1,#crc$R$L'));
                            REG27:
                                strcpy(ADR(WriteData),ADR('rdm,0,27,1,#crc$R$L'));
                            REG28:
                                strcpy(ADR(WriteData),ADR('rdm,0,28,1,#crc$R$L'));
                            REG29:
                                strcpy(ADR(WriteData),ADR('rdm,0,29,1,#crc$R$L'));
                            REG30:
                                strcpy(ADR(WriteData),ADR('rdm,0,30,1,#crc$R$L'));
                            REG31:
                                strcpy(ADR(WriteData),ADR('rdm,0,31,1,#crc$R$L'));
                            REG32:
                                strcpy(ADR(WriteData),ADR('rdm,0,32,1,#crc$R$L'));
                            REG33:
                                strcpy(ADR(WriteData),ADR('rdm,0,33,1,#crc$R$L'));
                        END_CASE
                        CommandReady:=TRUE;
                        StepREAD		:=	OPEN;
                    ELSE
                        Error   		:=	1;
                        ErrorID 		:=	rfidError_read_wrongRegNr; (* wrong register number*)
                        Busy    		:=	0;
                        CommandReady	:=	0;
                        TypeOK			:=	FALSE;
                    END_IF
                END_IF
                IF CommandReady	= 1 THEN
                    CASE StepREAD OF
                        OPEN:
                            FrameXOpenStruct.mode:=ADR('/RIT=200 ');
                            FrameXOpenStruct(enable := 1,device := Ident);
                            status.XOPEN 			:= FrameXOpenStruct.status;
                            IF (status.XOPEN = 0) THEN
                                StepREAD            := WRITE ;
                                FrameXOpenStruct.enable:=FALSE;
                            ELSE
                                StepREAD            := OPEN ;
                                Error               := TRUE;
                                ErrorID             := status.XOPEN;
                                Busy                := 0;
                                FrameXOpenStruct.enable:=FALSE;
                            END_IF
                        WRITE:
                            FrameGetBufferStruct(enable:= 1, ident:= FrameXOpenStruct.ident);
                            sendbuffer				:= FrameGetBufferStruct.buffer;
                            sendbufferlength		:= FrameGetBufferStruct.buflng;
                            status.GetBuffer		:= FrameGetBufferStruct.status;
                            IF	(status.GetBuffer = 0)	THEN
                                memcpy(sendbuffer,ADR(WriteData),SIZEOF(WriteData));
                                FrameWriteStruct(enable := 1, ident := FrameXOpenStruct.ident, buffer := sendbuffer,buflng := strlen(ADR(WriteData)));
                                status.WRITE 		:=	FrameWriteStruct.status;
                                IF (status.WRITE <> 0) THEN
                                    FrameReleaseOutputBufferStruct(enable:=1,ident:=FrameXOpenStruct.ident,buffer:=sendbuffer,buflng:= strlen(ADR(WriteData)));
                                    status.RoBuffer			:= FrameReleaseOutputBufferStruct.status;
                                    IF	(status.RoBuffer <> 0)	THEN
                                        ErrorID := status.RoBuffer;
                                        FrameReleaseOutputBufferStruct.enable:=FALSE;
                                    END_IF
                                ELSE
                                    FrameWriteStruct.enable := 0;
                                    FrameGetBufferStruct.enable	:= 0;
                                    FrameReleaseOutputBufferStruct.enable := 0;
                                    StepREAD			:=	READ;
                                END_IF
                            ELSE
                                ErrorID 		:= status.GetBuffer;
                                Error   		:= 1;
                                Busy    		:= 0;
                                StepREAD		:= OPEN;
                                TypeOK			:= FALSE;
                                CommandReady	:=	0;
                                FrameGetBufferStruct.enable	:= 0;
                            END_IF

                        READ:
                            FrameReadStruct(enable := 1,ident:=FrameXOpenStruct.ident);
                            ReadBuffer       	:=	FrameReadStruct.buffer;
                            ReadBufferLength	:=	FrameReadStruct.buflng;
                            status.READ      	:=	FrameReadStruct.status;
                            IF  (status.READ = 0)  THEN
                                memset(ADR(ReadData),0,SIZEOF(ReadData));
                                memcpy(ADR(ReadData),ReadBuffer,ReadBufferLength);
                                FrameReadStruct.enable	:=	0;
                                FrameReleaseBufferStruct(enable:=1, ident:=FrameXOpenStruct.ident, buffer:=ReadBuffer,buflng:=ReadBufferLength);
                                status.ReleaseBuffer	:=	FrameReleaseBufferStruct.status;
                                IF (status.ReleaseBuffer	= 0) THEN
                                    FrameReleaseBufferStruct.enable	:=	0;
                                    AN[0]	:= ReadData[0];
                                    AN[1]	:= ReadData[1];
                                    AN[2]	:= ReadData[2];
                                    IF (memcmp(ADR(AN),ADR('ack'),3) = 0) THEN
                                        IF ReadBufferLength <> 22 THEN
                                            StepREAD		:=	OPEN;
                                            Error       	:=	1;
                                            ErrorID      	:=	rfidError_read_failed ; (* unknow answer *)
                                            Busy         	:=	0;
                                            CommandReady	:=	0;
                                            TypeOK			:=	FALSE;
                                        ELSE
                                            StepREAD    :=	DATAREAD;
                                        END_IF
                                    ELSIF	(memcmp(ADR(AN),ADR('nak'),3) = 0)	THEN
                                        ERROR[0]	:=	ReadData[6];
                                        ERROR[1]	:=	ReadData[7];
                                        ERROR[2]	:=	ReadData[8];
                                        StepREAD		:=	OPEN;
                                        Error       	:=	1;
                                        ErrorID      	:=	atoi(ADR(ERROR)) ;
                                        Busy         	:=	0;
                                        CommandReady	:=	0;
                                        TypeOK			:=	FALSE;
                                    ELSE
                                        StepREAD		:=	OPEN;
                                        Error       	:=	1;
                                        ErrorID      	:=	rfidError_read_failed ; (* unknow answer *)
                                        Busy         	:=	0;
                                        CommandReady	:=	0;
                                        TypeOK			:=	FALSE;
                                    END_IF
                                ELSE
                                    StepREAD		:=	OPEN;
                                    Error       	:=	1;
                                    ErrorID      	:=	status.ReleaseBuffer ;
                                    Busy         	:=	0;
                                    CommandReady	:=	0;
                                    TypeOK			:=	FALSE;
                                END_IF
                            ELSE
                                memset(ADR(ReadData),0,SIZEOF(ReadData));
                            END_IF
                        DATAREAD:
                            memset(ADR(data),0,SIZEOF(data));
                            data[0] 	 	:=	ReadData[6];
                            data[1] 	 	:=	ReadData[7];
                            data[2] 	 	:=	ReadData[8];
                            data[3] 	 	:=	ReadData[9];
                            data[4] 	 	:=	ReadData[10];
                            data[5] 	 	:=	ReadData[11];
                            data[6] 	 	:=	ReadData[12];
                            data[7] 	 	:=	ReadData[13];
                            Data			:=	ADR(data);
                            Done         	:=	1;
                            Busy         	:=	0;
                            CommandReady	:=	0;
                            StepREAD     	:=	OPEN;
                            TypeOK			:=	FALSE;
                    END_CASE
                END_IF
            END_IF
        END_IF
    ELSE
        Busy:=0;
        Done:=0;
        Error:=0;
        ErrorID:=0;
        StepREAD:= 0;
        StepType:= 0;
    END_IF
END_FUNCTION_BLOCK
```

### Program Logical/Program/Linka/Main (IEC)

#### Main.st - Init, cyclic, exit code
```iecst
PROGRAM _INIT

    Linka.PAR.IndexModelu:= 1;
    CasCakaniaNaDruhePracovisko:= 120000;

END_PROGRAM

PROGRAM _CYCLIC

    //Volba modelu//
    IF Linka.STAV.Vypnuta THEN
        IF Linka.PAR.IndexModelu = 0 THEN
            Linka.PAR.ZvolenyModel:= '4F';
        ELSIF Linka.PAR.IndexModelu = 1 THEN
            Linka.PAR.ZvolenyModel:= '5F';
        ELSIF Linka.PAR.IndexModelu = 2 THEN
            Linka.PAR.ZvolenyModel:= '5H';
        END_IF
    END_IF

    //Volanie podprogramov//
    ProfinetKomunikaciaCU;

    (*Pri zmene modelu kontrolovat či sú vymenené prípravky na testeroch inač nepovoliť spustenie výroby*)

    //**************************Zmena času a dátumu***************************************//
    IF Vizu.NastavCasPLC THEN
        DTSetTime_0.enable:= TRUE;
        DTSetTime_0.DT1:= Vizu.ZadanyCasPLC;
        DTSetTime_0();
    END_IF

    IF DTSetTime_0.status = 0 THEN
        Vizu.NastavCasPLC:= FALSE;
        DTSetTime_0.enable:= FALSE;
        DTSetTime_0();
    END_IF

    //**********************Načítanie času a dátumu do vizualizácie**************************//
    DTGetTime_0.enable:= TRUE;
    Vizu.AktualnyCasPLC:= DTGetTime_0.DT1;
    DTGetTime_0();

    //**************************Stav linka vypnuta********************************************//
    IF P1_Pracovisko.STAV.Automat THEN
        Linka.STAV.Vypnuta:= FALSE;
    ELSIF P2_Pracovisko.STAV.Automat THEN
        Linka.STAV.Vypnuta:= FALSE;
    ELSIF P3_Pracovisko.STAV.Automat THEN
        Linka.STAV.Vypnuta:= FALSE;
    ELSIF P4_Pracovisko.STAV.Automat THEN
        Linka.STAV.Vypnuta:= FALSE;
    ELSE
        Linka.STAV.Vypnuta:= TRUE;
    END_IF

    //***************************Stav linka po inicializacii********************************************//
    IF NOT P1_Pracovisko.STAV.PoINIT THEN
        Linka.STAV.PoINIT:= FALSE;
    ELSIF NOT P2_Pracovisko.STAV.PoINIT THEN
        Linka.STAV.PoINIT:= FALSE;
    ELSIF NOT P3_Pracovisko.STAV.PoINIT THEN
        Linka.STAV.PoINIT:= FALSE;
    ELSIF NOT P4_Pracovisko.STAV.PoINIT THEN
        Linka.STAV.PoINIT:= FALSE;
    ELSE
        Linka.STAV.PoINIT:= TRUE;
    END_IF

    //**************************Stav linka prazdna********************************************//
    IF NOT P1_StoperSrobovania.IN.PritomnostPaletky_S16 AND
        NOT P1_AkumulacnyStoper.IN.PritomnPaletky_IS45 AND
        NOT P2_StoperZaklTesnenia.IN.PritomnostPaletky_S6 AND
        NOT P2_StoperMaticovacky.IN.PritomnostPaletky_S7 AND
        NOT P2_StoperSrobovania.IN.PritomnostPaletky_S8 AND
        NOT P2_StoperZvarania.IN.PritomnostPaletky_S9 AND
        NOT P3_StoperSrobovania.IN.PritomnostPaletky_S22 AND
        NOT P3_AkumulacnyStoper.IN.PritomnPaletky_IS65 AND
        NOT P3_LeakageTestA.IN.PritomnostPaletky_S23 AND
        NOT P3_LeakageTestB.IN.PritomnostPaletky_S24 AND
        NOT P4_FunkcnyTestA.IN.PritomnostPaletky_S10 AND
        NOT P4_FunkcnyTestB.IN.PritomnostPaletky_S11 AND
        NOT P4_Etiketovacka.IN.PritomnostPaletky_S12 AND
        NOT P4_Vytah.IN.PritomnostPaletky_S13 THEN
        Linka.STAV.LinkaPrazdna:= TRUE;
    ELSE
        Linka.STAV.LinkaPrazdna:= FALSE;
    END_IF

    //**************************Režim vyprázdnenia linky*******************************************//
    Linka.VyprazdnenieLinky;

    //**************************Zber fotiek do adresara DMP**************************************//
    Linka.ZberFotiek;

END_PROGRAM

PROGRAM _EXIT
	(* Insert code here *)

END_PROGRAM
```

#### Variables.var - Local variables
```iecst
VAR
	T0_test : TON;
	timerString : STRING[255];
	timerREAL : REAL;
	Cas : TON;
	timerSekundyREAL : REAL;
	CasKontrolyVyprazdnenia : TON;
	CasKontrolyTestovania : TON;
END_VAR
```
